// TwinCAT 3 PLC project Area2
// ProgramVersion: 3.1.4023.0
// libraries:
//   Tc2_DataExchange, * (Beckhoff Automation GmbH)
//   Tc2_MC2, * (Beckhoff Automation GmbH)
//   Tc2_Standard, * (Beckhoff Automation GmbH)
//   Tc2_System, * (Beckhoff Automation GmbH)
//   Tc2_TcpIp, * (Beckhoff Automation GmbH)
//   Tc2_Utilities, * (Beckhoff Automation GmbH)
//   Tc3_BA_Common, * (Beckhoff Automation GmbH)
//   Tc3_Database, * (Beckhoff Automation GmbH)
//   Tc3_JsonXml, * (Beckhoff Automation GmbH)
//   Tc3_Module, * (Beckhoff Automation GmbH)
//   Tc3_PackML_V2, * (Beckhoff Automation GmbH)
// project tree:
//   COMMs_ADS/ AdsClient.TcPOU, AdsHandle.TcPOU
//   COMMs_ADS/PROTOTYPE/ AdsClient_1.TcPOU, AdsHandle_1.TcPOU (not stored)
//   COMMs_TCP/ TcpServer1Vision.TcPOU (not stored)
//   COMMs_TCP/Types/ DUT.TcDUT (not stored), TcpData.TcDUT, TcpDataQueue.TcPOU (not stored)
//   DUTs/Enums/ E_PMLCustomUnitMode.TcDUT, InsertionDirection.TcDUT (not stored), SectionEnum.TcDUT (not stored), SectionTask.TcDUT, ConveyorMode.TcDUT (not stored), Cover.TcDUT, EventsEnum.TcTLEO (not stored), MaterialEnums.TcDUT (not stored), MaterialType.TcDUT, Surface.TcDUT (not stored)
//   DUTs/Enums/Materials/ Cardboard.TcDUT (not stored), Chipboard.TcDUT (not stored), CornerGuard.TcDUT (not stored), WoodBunk.TcDUT (not stored)
//   DUTs/Enums/Robot Tasks/ A22.TcDUT, A21.TcDUT
//   DUTs/Hardware/ A21ToolStorage.TcDUT (not stored), ConveyorLSC.TcPOU (not stored), ConveyorSC.TcPOU, FoldingMachine.TcDUT (not stored), Conveyor.TcPOU (not stored)
//   DUTs/Hardware/Big Machines/ StrapMachine.TcPOU, WrapMachine.TcPOU
//   DUTs/Hardware/Insertion Package/Drives/ AirPiston.TcPOU (not stored), ClearLinkMC.TcPOU (not stored), ServoNC.TcPOU (not stored), SimplePiston.TcPOU
//   DUTs/Hardware/Insertion Package/ Homing.TcDUT, Insertion.TcPOU, SuctionPad.TcDUT (not stored)
//   DUTs/Hardware/Insertion Package/Prototypes/ FBA_Drive.TcPOU, FBA_TrifectaDrive.TcPOU (not stored), I_ContinuousDrive.TcIO, I_Drive.TcIO (not stored), I_EncodedDrive.TcIO (not stored), I_PositionalDrive.TcIO
//   DUTs/Hardware/Material Holders/ MaterialHolder.TcPOU, MaterialSlot.TcDUT, SkidMagazine.TcPOU (not stored), StagingTable.TcPOU (not stored)
//   DUTs/Hardware/Robots/ KukaRobot.TcPOU, RobotA21.TcPOU, RobotA22.TcPOU
//   DUTs/ ONE_BIT.TcDUT (not stored), VisionFrame.TcDUT (not stored), VisionSuite.TcDUT (not stored)
//   COMMs_ADS/Types/ AdsSocket.TcPOU (not stored), AdsDataQueue.TcPOU (not stored), AdsData.TcDUT (not stored)
//   DUTs/Bundle/ Bundle.TcDUT, CardboardMaterial.TcDUT (not stored), Interval.TcDUT (not stored), Material.TcDUT (not stored), PositionMaterials.TcDUT (not stored)
//   DUTs/Containers/ DynamicQueue.TcPOU (not stored), PtrQueue.TcPOU (not stored), IntQueue.TcPOU, Queue.TcPOU (not stored), StringQueue.TcPOU
//   EventLogging/ EventLogger.TcIO (not stored), SqlDatabaseAccessor.TcPOU (not stored)
//   / GlobalTextList.TcGTLO, PlcTask.TcTTO (not stored)
//   GVLs/ Conveyors.TcGVL, GVL.TcGVL, Hardware_A21.TcGVL, Hardware_A22.TcGVL, Hardware_A23.TcGVL, Hardware_A24.TcGVL (not stored), Hardware_A25.TcGVL (not stored), Misc.TcGVL (not stored), Param.TcGVL
//   POUs/ CallHardware.TcPOU, ConveyorControlUnit.TcPOU, MAIN.TcPOU
//   POUs/Helper Functions/Document/ CreateJsonDocumentManual.TcPOU, CreateJsonDocumentAuto.TcPOU (not stored), FrameIsValid.TcPOU (not stored), VisionJsonParser.TcPOU (not stored)
//   POUs/Helper Functions/General/ BufferIsEmpty.TcPOU (not stored), BundleIsValid.TcPOU, InRange.TcPOU (not stored), PositionIsValid.TcPOU, TimestructToString.TcPOU (not stored)
//   POUs/Helper Functions/Hardware Modules/ InsertionQuality.TcPOU (not stored), SetSuctions.TcPOU (not stored), SetSuctionsPtrArr.TcPOU (not stored), SetupHardware.TcPOU, SuctionQuality.TcPOU (not stored)
//   POUs/Helper Functions/Material Functions/ GetPositionMasterLength.TcPOU (not stored), GetMaterialLength.TcPOU (not stored), MatchesMaterialType.TcPOU (not stored)
//   POUs/Helper Functions/Other/ ForceSetLifterConveyors.TcPOU (not stored), SizeCheck.TcPOU (not stored)
//   POUs/Helper Functions/Utility/ AddToStringArray.TcPOU (not stored), DataIsEmtpy.TcPOU, CleanStringsArray.TcPOU, IntegerBitAccess.TcPOU, IntegerToBoolArray.TcPOU (not stored), JoinStrings.TcPOU (not stored), WithinTolerance.TcPOU
//   Sections/A21a - Chipboard/AOIs/ AOI_LoadChipboard.TcPOU
//   Sections/A21a - Chipboard/ ChipboardEx.TcPOU
//   Sections/A21b - Wood Bunk/AOIs/ AOI_LoadWoodBunk.TcPOU, AOI_StageWoodBunk.TcPOU, AOI_StagingTemplate.TcPOU, AOI_WoodBunkAlarms.TcPOU (not stored)
//   Sections/A21b - Wood Bunk/ WoodBunkEx.TcPOU
//   Sections/Abstract/ SectionEx.TcPOU
// real-time tasks:
//   TASK PlcTask: cycle T#10ms, priority 20, ADS port 350

// ---- COMMs_TCP/Types/TcpData.TcDUT
{attribute 'enable_dynamic_creation'}
TYPE TcpData :
UNION
	binaryData : ARRAY[0..1000] OF BYTE; //contents
	toString : STRING(1000);
END_UNION
END_TYPE

// ---- DUTs/Enums/E_PMLCustomUnitMode.TcDUT
//{attribute 'qualified_only'}
//{attribute 'strict'}
TYPE E_PMLCustomUnitMode :
(
	ePMLCustomUnitMode_Invalid := 0, //no mode
	ePMLCustomUnitMode_Production := 1, //normal automatic production
	ePMLCustomUnitMode_Maintenance := 2, //testing operational improvements
	ePMLCustomUnitMode_Manual := 3, //commissioning
	
	ePMLCustomUnitMode_SemiAuto := 4, //same state machine as production, but uses an execute signal to advance to next step
	
	size
)DINT;
END_TYPE
(*
this enum adds on to E_PMLProtectedUnitMode with additional modes
can be used by a combobox on the HMI to select a mode

all modes used in the program need to be configured using PML_UnitModeConfig
*)

// ---- DUTs/Enums/Robot Tasks/A22.TcDUT
{attribute 'qualified_only'}
{attribute 'to_string'}
//{attribute 'strict'}
TYPE A22 :
(
	IDLE,
	
	LOAD_CARDBOARD_TOP, //flat cardboards
	LOAD_CARDBOARD_BOTTOM,
	LOAD_CARDBOARD_SIDE,
	REMOVE_CARDBOARD_TOP,
	REMOVE_CARDBOARD_BOTTOM,
	REMOVE_CARDBOARD_SIDE,
	
	TRANSFER_TO_BENDER := 9, //corner cardboards
	TRANSFER_TO_OVERHEAD,
	REMOVE_CARDBOARD_FROM_BENDER,
	LOAD_BENDER_TO_UPPER_CORNER,
	LOAD_BENDER_TO_LOWER_CORNER,
	LOAD_OVERHEAD_TO_UPPER_CORNER,
	LOAD_OVERHEAD_TO_LOWER_CORNER,
	
	REMOVE_CARDBOARD_UPPER_CORNER,
	REMOVE_CARDBOARD_LOWER_CORNER,
	REMOVE_CARDBOARD_OVERHEAD := 18,
	
	LOAD_CORNER_GUARD_UPPER := 20, //corner guards
	LOAD_CORNER_GUARD_LOWER,
	REMOVE_CORNER_GUARD_UPPER,
	REMOVE_CORNER_GUARD_LOWER,
	
	size
);
END_TYPE

// ---- DUTs/Hardware/Insertion Package/Homing.TcDUT
{attribute 'qualified_only'}
{attribute 'strict'}
TYPE Homing :
(
	IDLE,
	
	START,
	RETRY,
	
	STOP,
	SET,
	DONE,
	
	size
);
END_TYPE
(*
general homing sequence:
	on drive.homingSequence() call, home towards home sensor
	if home reached, set position and finish homing as usual
	if outer limit reached, traverse towards inner limit
		when inner limit reached, retry homing
*)

// ---- DUTs/Hardware/Material Holders/MaterialSlot.TcDUT
TYPE MaterialSlot :
STRUCT
	material : STRING;
	occupied AT %I* : BOOL;
END_STRUCT
END_TYPE

// ---- DUTs/Enums/Robot Tasks/A21.TcDUT
{attribute 'qualified_only'}
//{attribute 'strict'}
{attribute 'to_string'}
TYPE A21 :
(
	IDLE,
	STAGE_BUNK,
	REMOVE_BUNK_FROM_STAGE,
	
	LOAD_BUNK_TOP := 4,
	LOAD_BUNK_SIDE,
	LOAD_BUNK_BOTTOM,
	REMOVE_BUNK_TOP,
	REMOVE_BUNK_SIDE,
	REMOVE_BUNK_BOTTOM,
	
	//GET_CHIPBOARD_FROM_SKID := 11,
	//OFFLOAD_CHIPBOARD,
	PLACE_CHIPBOARD_TOP := 13,
	PLACE_CHIPBOARD_BOTTOM,
	REMOVE_CHIPBOARD_TOP,
	REMOVE_CHIPBOARD_BOTTOM,
	
	FIX_CHIPBOARD_ORIENTATION := 19,
	
	//testing only
	MOVE_HOME := 21,
	MOVE_POSITION1,
	MOVE_POSITION2,
	MOVE_UP,
	MOVE_DOWN,
	
	DIRECT_BUNK_TOP := 27,
	DIRECT_BUNK_SIDE,
	DIRECT_BUNK_BOTTOM,
	
	INSPECT_BUNK := 31,
	INSPECT_CHIPBOARD,
	
	TOOL_CHANGE_BUNK := 34,
	TOOL_CHANGE_CHIPBOARD,
	
	size
);
END_TYPE

// ---- DUTs/Bundle/Bundle.TcDUT
{attribute 'enable_dynamic_creation'}
TYPE Bundle :
STRUCT
	id : STRING;
	weight : REAL;
	
	length : INT;
	width : INT;
	height : INT;
	
	pieces : INT;
	layers : INT;
	piecesPerLayer : INT;
	
	extrusionWeight : INT;
	extrusionHeight : INT;
	extrusionWidth : INT;
	
	//if a process is true, send it to the correct area and turn it false when complete
	reqProcesses : ARRAY[0..3] OF BOOL;
	
	manRE, autoRE : BOOL; //repacking - coming soon
	manSS, autoSS : BOOL; //packaging
	
	currStep : USINT; //for runtime use only
	
	paperFront : BOOL;
	paperBack : BOOL;
	cardboardFront : BOOL;
	cardboardBack : BOOL;
	
	paperTop : ARRAY[0..GVL.maxPairs] OF Interval;
	paperLeft : ARRAY[0..GVL.maxPairs] OF Interval;
	paperRight : ARRAY[0..GVL.maxPairs] OF Interval;
	paperBottom : ARRAY[0..GVL.maxPairs] OF Interval;
		
	cardboard : ARRAY[0..GVL.maxPairs] OF PositionMaterials;
	cardboardFolds : ARRAY[Surface.TOP_LEFT..Surface.BOTTOM_RIGHT] OF ARRAY[0..GVL.maxPairs] OF INT;
	
	topLeftFolds : ARRAY[0..GVL.maxPairs] OF INT;
	topRightFolds : ARRAY[0..GVL.maxPairs] OF INT;
	bottomLeftFolds : ARRAY[0..GVL.maxPairs] OF INT;
	bottomRightFolds : ARRAY[0..GVL.maxPairs] OF INT;
	
	cornerGuard : ARRAY[0..GVL.maxPairs] OF PositionMaterials;
	
	chipboard : ARRAY[0..GVL.maxPairs] OF PositionMaterials;
	woodBunk : ARRAY[0..GVL.maxPairs] OF PositionMaterials;
	
	cardboard_over_cornerGuard : BOOL;
	
	//for production log database
	timeStart : TIMESTRUCT;
	timeDone : TIMESTRUCT;
END_STRUCT
END_TYPE

// ---- DUTs/Enums/SectionTask.TcDUT
{attribute 'qualified_only'}
//{attribute 'strict'}
TYPE SectionTask :
(
	IDLE,
	ALIGNING,
	ACTIVE,
	CLEARING,
	COMPLETE,
	
	size
);
END_TYPE

// ---- DUTs/Enums/Cover.TcDUT
{attribute 'qualified_only'}
{attribute 'strict'}
TYPE Cover :
(
	FRONT,
	BACK,
	size
);
END_TYPE

// ---- DUTs/Enums/MaterialType.TcDUT
{attribute 'qualified_only'}
{attribute 'strict'}
TYPE MaterialType :
(
	PAPER,
	CARDBOARD,
	CORNER_GUARD,
	CHIPBOARD,
	WOOD_BUNK,
	size
);
END_TYPE

// ---- GVLs/Conveyors.TcGVL
//{attribute 'qualified_only'}
VAR_GLOBAL CONSTANT
	numConveyors : INT := 38;
END_VAR
VAR_GLOBAL
	conveyorsArr : ARRAY[1..numConveyors] OF POINTER TO ConveyorSC;
	
	A24_LRC_C02 	: Conveyor; //these conveyoors move bundles from A2.7 to A2.4
	A24_LRC_C04 	: Conveyor;
	A24_LRC_C06	 	: Conveyor;
	A24_LRC_C08 	: Conveyor;
	A24_LRC_C10 	: Conveyor;
	A24_LRC_C12 	: Conveyor;
	
	A24_SC_C01 		: ConveyorSC; //these conveyors move bundles on A2.4 forward down the cell
	A24_SC_C03 		: ConveyorSC;
	A24_SC_C05 		: ConveyorSC;
	A24_SC_C07 		: ConveyorSC;
	A24_SC_C09 		: ConveyorSC;
	A24_SC_C11 		: ConveyorSC;
	A24_SC_C13 		: ConveyorSC;
	
	A23_LSC_C14 	: ConveyorLSC;
	
	A22_SC_C15 		: ConveyorSC;
	A22_LSC_C16 	: ConveyorLSC;
	A22_LSC_C17 	: ConveyorLSC;
	
	A21_SC_C18 		: ConveyorSC;
	A21_LSC_C19 	: ConveyorLSC;
	A21_LSC_C20 	: ConveyorLSC;
	A21_LSC_C21 	: ConveyorLSC;
	
	A25_SC_C22 		: ConveyorSC;
	A25_LSC_C23 	: ConveyorLSC;
	A25_SC_C24 		: ConveyorSC;
	A25_LSLCC_C25 	: ConveyorLSC;
	A25_SC_C26 		: ConveyorSC;
	A25_LSLCC_C27 	: ConveyorLSC;
	A25_SC_C28 		: ConveyorSC;
	A25_LSC_C29 	: ConveyorLSC;
	A25_SC_C30 		: ConveyorSC;
	
	A25_SC_C31 		: ConveyorSC; //these conveyors move the bundle sideways onto the output buffers
	A25_SC_C32 		: ConveyorSC;
	A25_SC_C33 		: ConveyorSC;
	A25_SC_C34 		: ConveyorSC;
	A25_SC_C35 		: ConveyorSC;
	A25_SC_C36 		: ConveyorSC;
	A25_SC_C37 		: ConveyorSC;
	A25_SC_C38 		: ConveyorSC;
END_VAR

// ---- GVLs/GVL.TcGVL
{attribute 'qualified_only'}
VAR_GLOBAL CONSTANT
	maxPairs : USINT := 16;
	initArraySize : USINT := 4;
	maxQueue : INT := 16;
	
	nullPos : REAL := -1;
	
	numMaterials : INT := 32;
	allMaterials : ARRAY[0..numMaterials] OF Material := [
		(code := 'PAP28', width := 28, length := -1),
		
		(code := 'CAR20S', width := 20, length := 30),
		(code := 'CAR20M', width := 20, length := 45),
		(code := 'CAR20L', width := 20, length := 60),
		(code := 'CAR28S', width := 28, length := 30),
		(code := 'CAR28M', width := 28, length := 45),
		(code := 'CAR28L', width := 28, length := 60),
		
		(code := 'COR48', width := 1.5, length := 48),
		(code := 'COR96', width := 1.5, length := 96),
		
		(code := 'CIP18', width := 20, length := 18),
		(code := 'CIP54', width := 20, length := 54),
		
		(code := 'WDT20', width := 20, length := 2.5),
		(code := 'WDT22', width := 22, length := 2.5),
		(code := 'WDT28', width := 28, length := 2.5),
		
		(code := 'WDB20', width := 20, length := 2.5),
		(code := 'WDB22', width := 22, length := 2.5),
		(code := 'WDB28', width := 28, length := 2.5),
		
		(code := 'WDS08', width := 8, length := 2.5),
		(code := 'WDS10', width := 10, length := 2.5),
		(code := 'WDS12', width := 12, length := 2.5),
		(code := 'WDS14', width := 14, length := 2.5),
		(code := 'WDS8x8', width := 16, length := 2.5),
		(code := 'WDS8x10', width := 18, length := 2.5),
		(code := 'WDS20', width := 20, length := 2.5),
		(code := 'WDS22', width := 22, length := 2.5),
		(code := 'WDS12x12', width := 24, length := 2.5),
		(code := 'WDS12x14', width := 26, length := 2.5),
		(code := 'WDS28', width := 28, length := 2.5),
		(code := 'WDS20x10', width := 30, length := 2.5),
		(code := 'WDS20x12', width := 32, length := 2.5),
		
		(code := 'WDW20', width := 20, length := 6),
		(code := 'WDW22', width := 22, length := 6)]; //+1 null material

	//nullBundle : Bundle;
	
	//conveyorLength : REAL := 0;
	precisionTolerance : REAL := 0.05 * 25.4;
END_VAR
VAR_GLOBAL
	bundleOut : Bundle; //may or may not be used?
END_VAR

// ---- GVLs/Hardware_A21.TcGVL
//{attribute 'qualified_only'}
VAR_GLOBAL
	robot1 : RobotA21;
	robot2 : RobotA21;
	
	toolStorageA21Left : A21ToolStorage;
	toolStorageA21Right : A21ToolStorage;
	
	skidA21Left : SkidMagazine;
	skidA21Right : SkidMagazine;
	
	magazineA21Left : SkidMagazine;
	magazineA21Right : SkidMagazine;
	stagingTableLeft : StagingTable;
	stagingTableRight : StagingTable;
	
	strapperA21 : StrapMachine;
	
	horizontalDriveA21Left, horizontalDriveA21Right : AirPiston := (
		limitSensorDefaultState := FALSE,
		useBrake := FALSE);
	
	verticalDriveA21Left, verticalDriveA21Right : ClearLinkMC := (
		limitSensorDefaultState := TRUE, 
		homingDirectionOut := TRUE, //outwards (up)
		minPosition := 0,
		displacementPerRotation := 1,
		unitsPerPulse := 8000); //0.1x gearbox, 10 revs/pulse to compensate
		
	insertionA21left : Insertion;
	insertionA21Right : Insertion;
	
	pistonA21Bottom : SimplePiston;
	
	suctionA21Top : ARRAY[1..3] OF SuctionPad;
	suctionA21Left : ARRAY[1..4] OF SuctionPad;
	suctionA21Right : ARRAY[1..4] OF SuctionPad; 
	suctionA21Bottom : ARRAY[1..2] OF SuctionPad;
END_VAR
VAR_GLOBAL

	skidHmiA21Left, skidHmiA21Right AT %M* : ARRAY[1..2] OF MaterialSlot;
	magazineHmiA21Left, magazineHmiA21Right AT %M* : ARRAY[1..15] OF MaterialSlot;
	tableHmiA21Left, tableHmiA21Right : ARRAY[1..10] OF MaterialSlot;
END_VAR

// ---- GVLs/Hardware_A22.TcGVL
//{attribute 'qualified_only'}
VAR_GLOBAL
	robot3 : RobotA22;
	robot4 : RobotA22;
	
	benderA22Left : FoldingMachine;
	
	skidA22Left : SkidMagazine;
	skidA22Right : SkidMagazine;
	magazineA22Left : SkidMagazine;
	magazineA22Right : SkidMagazine;
	
	wrapperA22 : WrapMachine;
	overhead : STRING;
	
	horizontalDriveA22Left, horizontalDriveA22Right : ServoNC := (
		limitSensorDefaultState := TRUE);
		
	verticalDriveA22Left, verticalDriveA22Right : ClearLinkMC := (
		limitSensorDefaultState := TRUE, 
		homingDirectionOut := TRUE, //outwards (up)
		minPosition := (26*5 * 25.4),
		displacementPerRotation := 5,
		unitsPerPulse := 800); //800 counts = 1 rotation
		
	insertionA22Left : Insertion;
	insertionA22Right : Insertion;

	pistonA22Bottom : SimplePiston;
	
	(*
	each insertion suction array has 3 pads
	[1] - top/bottom
	[2] - corner
	[3] - side
	*)
	suctionA22TopLeft : ARRAY[1..3] OF SuctionPad;
	suctionA22TopRight : ARRAY[1..3] OF SuctionPad;
	suctionA22BottomLeft : ARRAY[1..3] OF SuctionPad; 
	suctionA22BottomRight : ARRAY[1..3] OF SuctionPad;
	
	suctionA22Bottom : ARRAY[1..2] OF SuctionPad;
END_VAR
VAR_GLOBAL //data arrays to be passed into material holder FBs - do not access directly
	skidHmiA22Left, skidHmiA22Right AT %M* : ARRAY[1...Cardboard.size-1] OF MaterialSlot;
	magazineHmiA22Left, magazineHmiA22Right AT %M* : ARRAY[1..CornerGuard.size-1] OF MaterialSlot;
END_VAR

// ---- GVLs/Hardware_A23.TcGVL
//{attribute 'qualified_only'}
VAR_GLOBAL
	//robot5 : RobotA23;
	//robot6 : RobotA23;
	
	//6 ClearLinkMC
	//3 or 4 ServoNC
	
	wrapperA23 : WrapMachine;
END_VAR

// ---- GVLs/Param.TcGVL
{attribute 'qualified_only'}
VAR_GLOBAL CONSTANT
END_VAR

// ---- DUTs/Hardware/Insertion Package/Prototypes/I_ContinuousDrive.TcIO
INTERFACE I_ContinuousDrive EXTENDS I_Drive

METHOD ABSTRACT moveContinuous : BOOL
VAR_INPUT
	direction : MC_Direction;
END_VAR
END_METHOD

END_INTERFACE

// ---- DUTs/Hardware/Insertion Package/Prototypes/I_PositionalDrive.TcIO
INTERFACE I_PositionalDrive EXTENDS I_Drive

{attribute 'monitoring':='call'}
PROPERTY AtOuterLimit : BOOL
GET
END_GET
END_PROPERTY

PROPERTY CurrentPosition : LREAL
GET
END_GET
SET
END_SET
END_PROPERTY

METHOD ABSTRACT moveAbsolute : BOOL
VAR_INPUT
	newTarget : LREAL; 
END_VAR
END_METHOD

METHOD ABSTRACT moveRelative : BOOL
VAR_INPUT
	distance : LREAL;
END_VAR
END_METHOD

PROPERTY TargetPosition : LREAL
GET
END_GET
SET
END_SET
END_PROPERTY

END_INTERFACE

// ---- DUTs/Hardware/ConveyorSC.TcPOU
FUNCTION_BLOCK ConveyorSC
VAR_INPUT
	bEnable : BOOL;
END_VAR
VAR_OUTPUT
	trueMode : ConveyorMode;
	requestedMode : ConveyorMode;
	
	error AT %I* : BOOL;
	position AT %I* : REAL;
	velocity AT %I* : REAL;
END_VAR
VAR
	enable AT %Q* : BOOL := TRUE;
	direction AT %Q* : BOOL; //FALSE = forward, TRUE = backward
	pulse AT %Q* : BOOL;
	reset AT %Q* : BOOL;
	
	sensorEntry AT %I* : BOOL := TRUE;
	sensorExit AT %I* : BOOL;
END_VAR
VAR
	//nextConveyor : POINTER TO ConveyorSC;
	//prevConveyor : POINTER TO ConveyorSC;
	
	pulser : TP; //pulses are assumed to be low-high-low
END_VAR
VAR_STAT CONSTANT
	pulseWidth : TIME := T#50MS;
END_VAR

enable := bEnable;

override();

sequence();

METHOD backward : BOOL
VAR_INPUT
END_VAR
END_METHOD

METHOD forward : BOOL
VAR_INPUT
END_VAR
END_METHOD

{attribute 'monitoring' := 'call'}
PROPERTY IsOccupied : BOOL
GET
IsOccupied := sensorExit OR sensorEntry;
END_GET
END_PROPERTY

METHOD join : BOOL
VAR_INPUT
	conveyor : POINTER TO ConveyorSC;
END_VAR
//nextConveyor := conveyor;
//conveyor^.prevConveyor := THIS;
END_METHOD

METHOD PROTECTED override : BOOL
VAR_INPUT
END_VAR
END_METHOD

METHOD reset : BOOL
VAR_INPUT
END_VAR
position := 0;
velocity := velocity; //no change
END_METHOD

METHOD PROTECTED sequence : BOOL
VAR_INPUT
END_VAR
direction := (trueMode = ConveyorMode.BACKWARD); //set direction bit

pulser(IN:= , PT:= pulseWidth, Q=> pulse, ET=> );
pulser.IN := 
	enable AND 
	NOT error AND 
	NOT reset AND 
	(trueMode = ConveyorMode.FORWARD OR trueMode = ConveyorMode.BACKWARD)
	AND pulser.Q; //ends pulse itself
END_METHOD

METHOD setMode : BOOL
VAR_INPUT
	mode : ConveyorMode;
END_VAR
trueMode := mode;
END_METHOD

METHOD setRequest : BOOL
VAR_INPUT
	newRequest : ConveyorMode;
END_VAR
requestedMode := newRequest;
END_METHOD

METHOD target : BOOL
VAR_INPUT
	targetPosition : REAL;
END_VAR
END_METHOD

END_FUNCTION_BLOCK

// ---- DUTs/Hardware/Robots/RobotA21.TcPOU
FUNCTION_BLOCK RobotA21 EXTENDS KukaRobot
VAR_OUTPUT //from outputs array
	{warning disable C0195}
	taskID : A21;
	param1 : INT;
	param2 : INT;
	Xmm : INT;
	Ymm : INT;
	Zmm : INT;
	angle : INT;
	stagingOccupancy : INT;
	insertionSuctionStatus : INT;
	magazineStatus : INT; //unused
	inspectionValue : INT;
	
	strapSafetyOut : BOOL;
END_VAR
VAR_OUTPUT //from inputs array
	tool : SectionEnum := SectionEnum.WOOD_BUNK;
	suspendedMaterial : STRING;
	//gripper : EOAT := (id := SectionEnum.WOOD_BUNK, material := '');
	
	completedTask : A21;
	eoatDistance : INT;
	woodBunkAvailability : INT;
	chipboardAvailability : INT;
	materialAtHoldingPosition : INT;
	
	strapSafetyIn : BOOL;
END_VAR
VAR
	reservationEnum : SectionEnum;
	hmiTask : STRING;
	hmiTool : STRING;
END_VAR
(*
extends KukaRobot
assigns descriptive labels to each IO group from the array
additional section-specific methods to get/set IO groups
*)

(*
parameters - aliases to IO elements
command - full IO array
*)
{warning disable C0195}
SUPER^();

strapSafetyOut := NOT strapperA21.enable AND NOT strapperA21.execute;
outputs[8].15 := strapSafetyOut;

outputs[1] := taskID;
outputs[2] := param1;
outputs[3] := param2;
outputs[4] := Xmm;
outputs[5] := Ymm;
outputs[6] := Zmm;
outputs[7] := angle;
outputs[8] := stagingOccupancy;
outputs[9] := insertionSuctionStatus;
outputs[10] := magazineStatus;
outputs[11] := inspectionValue;

outputs[8].15 := strapSafetyOut;

refreshParameters();

reservationEnum := reservation;
IF reservationEnum = SectionEnum.NULL_SECTION THEN
	hmiReservation := 'N/A';
ELSE
	hmiReservation := TO_STRING(reservationEnum);
END_IF

hmiTask := TO_STRING(taskID);
hmiTool := TO_STRING(tool);

{attribute 'monitoring' := 'call'}
PROPERTY Busy : BOOL
GET
VAR
	//emptyOutput : ARRAY[1..50] OF INT;
END_VAR
//Busy stays TRUE until outputs are cleared AND completed task has elapsed
//Ready is always inverse of Busy
refreshParameters();

Busy := taskID <> 0 OR completedTask <> 0;
END_GET
END_PROPERTY

METHOD changeEOAT : BOOL
VAR_INPUT
	targetTool : SectionEnum;
END_VAR
setGroup(group := 1, value := A21.TOOL_CHANGE_CHIPBOARD);
setGroup(group := 1, value := A21.TOOL_CHANGE_BUNK);

changeEOAT := tool = targetTool;
END_METHOD

METHOD clearCommand : BOOL
VAR_INPUT
END_VAR
SUPER^.clearCommand();

refreshParameters();
END_METHOD

{attribute 'monitoring' := 'call'}
PROPERTY Done : BOOL
GET
refreshParameters();

Done :=
	completedTask = taskID AND
	taskID <> 0 AND
	completedTask <> 0;
END_GET
END_PROPERTY

{attribute 'monitoring' := 'call'}
PROPERTY HoldMaterial : STRING
GET
HoldMaterial := suspendedMaterial;
END_GET
SET
suspendedMaterial := HoldMaterial;
END_SET
END_PROPERTY

{attribute 'monitoring' := 'call'}
PROPERTY Ready : BOOL
GET
refreshParameters();

Ready := taskID = 0 AND completedTask = 0;
END_GET
END_PROPERTY

METHOD PRIVATE refreshParameters : BOOL
VAR_INPUT
END_VAR
{warning disable C0196}
taskID := outputs[1];
param1 := outputs[2];
param2 := outputs[3];
Xmm := outputs[4];
Ymm := outputs[5];
Zmm := outputs[6];
angle := outputs[7];
stagingOccupancy := outputs[8];
insertionSuctionStatus := outputs[9];
magazineStatus := outputs[10]; //unused
inspectionValue := outputs[11];

completedTask := inputs[1];
eoatDistance := inputs[2];
woodBunkAvailability := inputs[3];
chipboardAvailability := inputs[4];
materialAtHoldingPosition := inputs[5];
//robotEOAT := inputs[6];

strapSafetyIn := inputs[4].15;
END_METHOD

METHOD setGroup : BOOL
VAR_INPUT
	group : INT;
	value : INT;
END_VAR
SUPER^.setGroup(group := group, value := value);

refreshParameters();
END_METHOD

METHOD setParameters : BOOL
VAR_INPUT
	newTaskID : INT;
	newParam1 : INT;
	newParam2 : INT;
	newXmm : INT;
	newYmm : INT;
	newZmm : INT;
	newAngle : INT;
	newStagingOccupancy : INT;
	newInsertionSuctionStatus : INT;
	newMagazineStatus : INT; //unused
	newInspectionValue : INT;
END_VAR
VAR_INPUT
	strapSafety : BOOL;
END_VAR
setGroup(group := 1, value := newTaskID);
setGroup(group := 2, value := newParam1);
setGroup(group := 3, value := newParam2);
setGroup(group := 4, value := newXmm);
setGroup(group := 5, value := newYmm);
setGroup(group := 6, value := newZmm);
setGroup(group := 7, value := newAngle);

newStagingOccupancy.15 := strapSafety;
setGroup(group := 8, value := newStagingOccupancy);

setGroup(group := 9, value := newInsertionSuctionStatus);
setGroup(group := 10, value := newMagazineStatus);
setGroup(group := 11, value := newInspectionValue);

refreshParameters();
END_METHOD

END_FUNCTION_BLOCK

// ---- DUTs/Hardware/Robots/KukaRobot.TcPOU
FUNCTION_BLOCK KukaRobot
VAR_OUTPUT
	forceStop AT %Q* : BOOL;
	resetSignal AT %Q* : BOOL;
	
	offline AT %I* : BOOL;
	operational : BOOL;
	reservation : INT := SectionEnum.NULL_SECTION;
	
	error : BOOL;
	errId : DINT;
	
	outputs AT %Q* : ARRAY[1..50] OF WORD;
	inputs AT %I* : ARRAY[1..20] OF WORD;
END_VAR
VAR
	hmiReservation : STRING;
END_VAR
(*
generic KUKA robot with 50 WORD outputs and 20 WORD inputs
includes minimal diagnostics to detect if robot is offline
robots should always be reserved before sending a task
*)

operational := NOT offline;

error := offline; //add any addition conditions with OR

//{attribute 'monitoring' := 'variable'}
{attribute 'monitoring' := 'call'}
PROPERTY Busy : BOOL
GET
END_GET
END_PROPERTY

METHOD clearCommand : BOOL
VAR_INPUT
END_VAR
MEMSET(ADR(outputs), 0, SIZEOF(outputs));
END_METHOD

//{attribute 'monitoring' := 'variable'}
{attribute 'monitoring' := 'call'}
PROPERTY Done : BOOL
GET
END_GET
END_PROPERTY

METHOD eStop : BOOL
VAR_INPUT
END_VAR
forceStop := TRUE;
eStop := TRUE;
END_METHOD

METHOD fullCommand : BOOL
VAR_INPUT
	newOutputs : REFERENCE TO ARRAY[1..50] OF WORD;
END_VAR
//IF NOT Busy THEN
	//RETURN;
//END_IF

outputs := newOutputs;
fullCommand := Done;

(*
CASE step OF
	SEND_COMMAND: //wait 1 cycle
		outputs := newOutputs;
		step := WAIT;
		
	WAIT:
		IF done THEN
			(*	
			IF NOT reset() THEN
				RETURN;
			END_IF
			
			step := 0;
			*)
			setCommandAndWait := TRUE;
		END_IF
		
END_CASE
*)
END_METHOD

{attribute 'monitoring' := 'call'}
PROPERTY Ready : BOOL
GET
END_GET
END_PROPERTY

METHOD release : BOOL
VAR_INPUT
	sectionReservation : SectionEnum;
END_VAR
IF reservation = sectionReservation THEN
	reservation := SectionEnum.NULL_SECTION;
	release := TRUE;
END_IF
END_METHOD

METHOD reserve : BOOL
VAR_INPUT
	reserveRequest : SectionEnum;
END_VAR
(*
this method exists because chipboard and wood bunk operations use the same robot
both sections need to check if the robot is open to commands before use
*)
IF Reserved AND reservation = reserveRequest THEN
	reserve := TRUE;

ELSIF NOT Reserved THEN
	reservation := reserveRequest;
	reserve := TRUE;

END_IF
END_METHOD

{attribute 'monitoring' := 'call'}
PROPERTY Reserved : BOOL
GET
Reserved := reservation <> SectionEnum.NULL_SECTION;
END_GET
END_PROPERTY

METHOD reset : BOOL
//resetSignal := TRUE;
//done := FALSE;

MEMSET(ADR(outputs), 0, SIZEOF(outputs));
(*
IF ready AND completedTask = 0 THEN
	resetSignal := FALSE;
	reset := TRUE;
END_IF
*)
END_METHOD

METHOD resume : BOOL
VAR_INPUT
END_VAR
forceStop := FALSE;

resume := NOT error AND errId = 0;
END_METHOD

METHOD setGroup : BOOL
VAR_INPUT
	group : INT;
	value : INT;
END_VAR
{warning disable C0195}
outputs[group] := value;
END_METHOD

END_FUNCTION_BLOCK

// ---- DUTs/Hardware/Big Machines/StrapMachine.TcPOU
FUNCTION_BLOCK StrapMachine
VAR_INPUT
	bEnable : BOOL;
END_VAR
VAR_OUTPUT
	enable AT %Q* : BOOL;
	execute AT %Q* : BOOL;
	reset AT %Q* : BOOL;
	
	error AT %I* : BOOL;
	ready AT %I* : BOOL;
	//busy (*AT %I**) : BOOL;
	done AT %I* : BOOL;
	home AT %I* : BOOL;
	
	timeout : BOOL;
	
	atBundleLevel AT %I* : BOOL;
END_VAR
VAR	
	holdPost : TON;
	timeoutDelay : TON;
	resetDelay : TP;
	
	start : BOOL;
	step : (SETUP, RUN, WAIT);
END_VAR
VAR_STAT CONSTANT
	maxDelay : TIME := T#30S;
	pulseWidth : TIME := T#500MS;
END_VAR

holdPost(IN:= , PT:= pulseWidth, Q=> , ET=> );
timeoutDelay(IN:= (step > 0), PT:= maxDelay, Q=> timeout, ET=> );

resetDelay(IN:= error AND NOT resetDelay.Q , PT:= pulseWidth, Q=> , ET=> );
reset := resetDelay.Q AND (resetDelay.ET > resetDelay.PT/2);

IF timeoutDelay.Q THEN
	timeoutDelay.IN := FALSE;
	timeout := TRUE;
	//busy := FALSE;
	
	start := FALSE;
	step := SETUP;
END_IF

enable := bEnable AND robot1.strapSafetyIn AND robot2.strapSafetyIn;

CASE step OF
	SETUP:
		IF error THEN
			enable := FALSE;
			execute := FALSE;
			RETURN;
		END_IF
		
		IF start AND enable (*AND ready*) THEN //strapping does not start if error
			start := FALSE;
			step := RUN;
		END_IF
	
	RUN:
		IF NOT execute THEN
			execute := TRUE;
			RETURN; //keeps execute TRUE for at least 1 cycle
		END_IF
		
		IF execute AND NOT ready (*AND NOT home*) THEN
			execute := FALSE;
			step := WAIT;
		END_IF
		
	WAIT: //due to the use of DC motors instead of stepper motors in the machine, a short delay is required before next strap
		IF home THEN
			holdPost.IN := TRUE;
			execute := FALSE;
			enable := FALSE;
		END_IF
		
		IF holdPost.Q THEN
			holdPost.IN := FALSE;
			step := 0;
		END_IF
		
END_CASE

(*
executePulse(IN:= , PT:= pulseTime, Q=> , ET=> );
execute := executePulse.IN AND NOT executePulse.Q;

IF executePulse.Q THEN
	executePulse.IN := FALSE;
END_IF


resetPulse(IN:= , PT:= pulseTime, Q=> , ET=> );
StrapMachineST.reset := resetPulse.IN AND NOT resetPulse.Q;

IF resetPulse.Q THEN
	executePulse.IN := FALSE;
END_IF

ready := enable AND NOT execute AND NOT StrapMachineST.reset AND NOT error AND home;
*)

METHOD clear : BOOL
VAR_INPUT
END_VAR
(*
reset should be continuously called until machine returns evidence that it is ready again
machine is expected to not respond to reset signals if it is already in an idle state
*)
END_METHOD

METHOD strap : BOOL
VAR_INPUT
END_VAR
//IF ready AND NOT busy AND NOT error THEN
	//busy := TRUE;
	//start := TRUE;
	//strap := TRUE;
//END_IF

start := TRUE;
END_METHOD

END_FUNCTION_BLOCK

// ---- DUTs/Hardware/Insertion Package/Insertion.TcPOU
FUNCTION_BLOCK Insertion //2d insertion that combines a slider (alignment) and screw (push)
VAR_INPUT
	enable : BOOL;
END_VAR
VAR_INPUT //interface references to existing drives
	slider : I_EncodedDrive;
	screw : I_ContinuousDrive;
END_VAR
VAR_OUTPUT
	contact AT %I* : BOOL;
	
	active : BOOL;
	error : BOOL;
	home : BOOL;
	
	homingComplete : BOOL;
	
	sliderPos : LREAL;
END_VAR
(*
this FB encapsulates 2 drives into a generic insertion machine
both drives should be declared externally in Hardware GVL as a concrete FB
Insertion instance should be declared and called in module scope, with the drives from Hardware GVL passed in by Interface reference
*)

homingComplete := slider.HomeSet AND screw.HomeSet;

active := slider.Active OR screw.Active;
error := slider.Error OR screw.Error;
home := slider.AtHome AND screw.AtHome;

sliderPos := slider.CurrentPosition;

METHOD align : BOOL
VAR_INPUT
	targetPos : REAL;
END_VAR
slider.moveAbsolute(newTarget := targetPos);
END_METHOD

METHOD homingSequence : BOOL
VAR_INPUT
END_VAR
IF NOT slider.homeSet THEN
	slider.homingSequence();
END_IF

IF NOT screw.homeSet THEN
	screw.homingSequence();
END_IF

homingSequence := homingComplete;
END_METHOD

METHOD press : BOOL
VAR_INPUT
END_VAR
screw.moveContinuous(direction := MC_Negative_Direction);
END_METHOD

METHOD release : BOOL
VAR_INPUT
END_VAR
screw.moveContinuous(direction := MC_Positive_Direction);
END_METHOD

METHOD reset : BOOL
VAR_INPUT
END_VAR
slider.reset();
screw.reset();
END_METHOD

METHOD stop : BOOL
VAR_INPUT
END_VAR
screw.stop();
slider.stop();
END_METHOD

METHOD toHome : BOOL
VAR_INPUT
END_VAR
slider.toHome();
screw.toHome();

toHome := slider.AtHome AND screw.AtHome;
END_METHOD

METHOD traverse : BOOL
VAR_INPUT
	direction : MC_Direction;
END_VAR
slider.moveContinuous(direction := MC_Negative_Direction);
END_METHOD

END_FUNCTION_BLOCK

// ---- DUTs/Hardware/Insertion Package/Drives/SimplePiston.TcPOU
FUNCTION_BLOCK SimplePiston
VAR_INPUT
	bEnable : BOOL;
END_VAR
VAR_OUTPUT
	pistonExtend AT %Q* : BOOL;
	pistonRetract AT %Q* : BOOL;
	
	extended AT %I* : BOOL;
	retracted AT %I* : BOOL;
	
	busy : BOOL;
END_VAR
VAR
	mode : (HOLD, IN, OUT);
END_VAR

IF
	NOT bEnable OR
	(retracted AND_THEN (pistonRetract OR mode = OUT)) OR
	(extended AND_THEN (pistonExtend OR mode = IN))
THEN
	mode := HOLD;
END_IF

CASE mode OF
	HOLD:
		pistonRetract := FALSE;
		pistonExtend := FALSE;
		
	IN:
		pistonRetract := FALSE;
		pistonExtend := TRUE;
	
	OUT:
		pistonRetract := TRUE;
		pistonExtend := FALSE;
	
END_CASE

busy := mode = IN OR mode = OUT;

METHOD extend : BOOL
VAR_INPUT
END_VAR
mode := IN;
END_METHOD

METHOD retract : BOOL
VAR_INPUT
END_VAR
mode := OUT;

retract := retracted;
END_METHOD

METHOD stop : BOOL
VAR_INPUT
END_VAR
pistonExtend := FALSE;
pistonRetract := FALSE;
mode := HOLD;
END_METHOD

END_FUNCTION_BLOCK

// ---- DUTs/Hardware/Robots/RobotA22.TcPOU
FUNCTION_BLOCK RobotA22 EXTENDS KukaRobot
VAR_OUTPUT //from outputs array
	taskID : A22;
	param1 : INT;
	param2 : INT;
	Xmm : INT;
	Ymm : INT;
	Zmm : INT;
	angle : INT;
	foldPosition0 : INT;
	foldPosition1 : INT;
END_VAR
VAR_OUTPUT //from inputs array
	tool : SectionEnum := SectionEnum.CARDBOARD_CORNERGUARD;
	suspendedMaterial : STRING;
	
	completedTask : A22;
	eoatDistance : INT;
	cardboardAvailability : INT;
	cornerGuardAvailability : INT;
	materialAtHoldingPosition : INT;
	//grp6
	//grp7
	
	wrapSafetyIn : BOOL;
	
END_VAR
VAR //HMI data
	reservationEnum : SectionEnum;
	hmiTask : STRING;
	hmiTool : STRING;
END_VAR

{warning disable C0195}
SUPER^();

outputs[1] := taskID;
outputs[2] := param1;
outputs[3] := param2;
outputs[4] := Xmm;
outputs[5] := Ymm;
outputs[6] := Zmm;
outputs[7] := angle;
outputs[8] := foldPosition0;
outputs[9] := foldPosition1;

refreshParameters();

reservationEnum := reservation;
IF reservationEnum = SectionEnum.NULL_SECTION THEN
	hmiReservation := 'N/A';
ELSE
	hmiReservation := TO_STRING(reservationEnum);
END_IF

hmiTask := TO_STRING(taskID);
hmiTool := TO_STRING(tool);

{attribute 'monitoring' := 'call'}
PROPERTY Busy : BOOL
GET
VAR
	//emptyOutput : ARRAY[1..50] OF INT;
END_VAR
//Busy stays TRUE until outputs are cleared AND completed task has elapsed
//Ready is always inverse of Busy
refreshParameters();

Busy := taskID <> 0 OR completedTask <> 0;
END_GET
END_PROPERTY

METHOD changeEOAT : BOOL
VAR_INPUT
	targetTool : SectionEnum;
END_VAR
//fill in IO here

changeEOAT := TRUE;
END_METHOD

METHOD clearCommand : BOOL
VAR_INPUT
END_VAR
SUPER^.clearCommand();

refreshParameters();
END_METHOD

{attribute 'monitoring' := 'call'}
PROPERTY Done : BOOL
GET
refreshParameters();

Done :=
	completedTask = taskID AND
	taskID <> 0 AND
	completedTask <> 0;
END_GET
END_PROPERTY

{attribute 'monitoring' := 'call'}
PROPERTY HoldMaterial : STRING
GET
HoldMaterial := suspendedMaterial;
END_GET
SET
suspendedMaterial := HoldMaterial;
END_SET
END_PROPERTY

{attribute 'monitoring' := 'call'}
PROPERTY Ready : BOOL
GET
refreshParameters();

Ready := taskID = 0 AND completedTask = 0;
END_GET
END_PROPERTY

METHOD PRIVATE refreshParameters : BOOL
VAR_INPUT
END_VAR
{warning disable C0196}
taskID := outputs[1];
param1 := outputs[2];
param2 := outputs[3];
Xmm := outputs[4];
Ymm := outputs[5];
Zmm := outputs[6];
angle := outputs[7];
foldPosition0 := outputs[8];
foldPosition1 := outputs[9];

completedTask := inputs[1];
(*
eoatDistance := inputs[2];
magazineAvailability := inputs[3];
chipboardSkidInPosition := inputs[4];
materialAtHoldingPosition := inputs[5];
//robotEOAT := inputs[6];

strapSafetyIn := inputs[4].15;
*)
END_METHOD

METHOD setGroup : BOOL
VAR_INPUT
	group : INT;
	value : INT;
END_VAR
SUPER^.setGroup(group := group, value := value);

refreshParameters();
END_METHOD

METHOD setParameters : BOOL
VAR_INPUT
	newTaskID : INT;
	newParam1 : INT;
	newParam2 : INT;
	newXmm : INT;
	newYmm : INT;
	newZmm : INT;
	newAngle : INT;
	newStagingOccupancy : INT;
	newInsertionSuctionStatus : INT;
	newMagazineStatus : INT; //unused
	newInspectionValue : INT;
END_VAR
setGroup(group := 1, value := newTaskID);
setGroup(group := 2, value := newParam1);
setGroup(group := 3, value := newParam2);
setGroup(group := 4, value := newXmm);
setGroup(group := 5, value := newYmm);
setGroup(group := 6, value := newZmm);
setGroup(group := 7, value := newAngle);

newStagingOccupancy.15 := NOT wrapperA22.enable AND NOT wrapperA22.execute;
setGroup(group := 8, value := newStagingOccupancy);

setGroup(group := 9, value := newInsertionSuctionStatus);
setGroup(group := 10, value := newMagazineStatus);
setGroup(group := 11, value := newInspectionValue);

refreshParameters();
END_METHOD

END_FUNCTION_BLOCK

// ---- DUTs/Hardware/Big Machines/WrapMachine.TcPOU
FUNCTION_BLOCK WrapMachine
VAR_OUTPUT
	error AT %I* : BOOL;
	ready AT %I* : BOOL;
	busy AT %I* : BOOL;
	done (*AT %I**) : BOOL;
	home AT %I* : BOOL;
	
	rotations AT %Q* : INT;
	execute AT %Q* : BOOL;
	enable AT %Q* : BOOL;
	reset AT %Q* : BOOL;
	
	timeout : BOOL;
	
	trayOccupied AT %I* : BOOL;
	overheadMaterial : STRING;
END_VAR
VAR
	holdPost : TON;
	delay : TON;
	
	start : BOOL;
	step : (SETUP, RUN, WAIT);
END_VAR
VAR_STAT CONSTANT
	pulseTime : TIME := T#100MS;
	holdTime : TIME := T#500MS;
	maxDelay : TIME := T#30S;
END_VAR

holdPost(IN:= , PT:= holdTime, Q=> , ET=> );
delay(IN:= step > 0, PT:= maxDelay, Q=> , ET=> );

IF delay.Q THEN
	delay.IN := FALSE;
	timeout := TRUE;
	busy := FALSE;
	step := SETUP;
END_IF

CASE step OF
	SETUP:
		busy := FALSE;
		IF error THEN
			reset := NOT reset;
			enable := FALSE;//NOT enable;
			
		ELSE
			reset := FALSE;
			enable := TRUE;
			
			IF start THEN
				start := FALSE;
				step := RUN;
			END_IF
			
		END_IF
	
	RUN:
		execute := TRUE;
		IF execute AND NOT home THEN
			execute := FALSE;
			step := WAIT;
		END_IF
		
	WAIT:
		IF home THEN
			holdPost.IN := TRUE;
			enable := FALSE;
			execute := FALSE;
		END_IF
		
		IF holdPost.Q THEN
			holdPost.IN := FALSE;
			done := TRUE;
			step := 0;
		END_IF
		
END_CASE

METHOD clear : BOOL
VAR_INPUT
END_VAR
(*
reset should be continuously called until machine returns evidence that it is ready again
machine is expected to not respond to reset signals if it is already in an idle state
*)
enable := FALSE;
execute := FALSE;

IF error THEN
	reset := NOT reset;
	clear := NOT error;

ELSE
	reset := FALSE;
	clear := TRUE;
	
END_IF
END_METHOD

{attribute 'monitoring' := 'call'}
PROPERTY Overhead : STRING
GET
Overhead := overheadMaterial;
END_GET
SET
overheadMaterial := Overhead;
END_SET
END_PROPERTY

METHOD wrap : BOOL
VAR_INPUT
	reqRotations : INT;
END_VAR
IF ready AND NOT busy AND NOT error THEN
	rotations := reqRotations;
	busy := TRUE;
	start := TRUE;
	wrap := TRUE;
END_IF
END_METHOD

END_FUNCTION_BLOCK

// ---- COMMs_ADS/AdsClient.TcPOU
PROGRAM AdsClient
VAR_INPUT
	ServerNetId			: STRING; 	(* Server AmsNetId *)
	ServerPort 			: UINT;	(* Server port number *)
END_VAR
VAR_OUTPUT
	bBusy				: BOOL;
	err					: BOOL;
	errid				: UDINT;
	
	localPrgName 		: STRING;
	localNetId 			: STRING;
	localPort 			: UINT;
	
	socketReady				: BOOL;
	
	remoteAccessPrefix	: STRING := 'AdsServer.area[2].';
END_VAR
VAR
	setupTimer 			: TON;
	
	handle 				: AdsHandle;
	numHandles 			: INT(0..maxHandles);
	
	setupStep 			: (SET_LOCAL_ENDPOINT, CLOSE_CONNECTIONS, SEND_CONNECTION_DATA, RECEIVE_SERVER_DATA, FINISH_SETUP);
	
	fbGetLocalAmsNetId	: FB_GetLocalAmsNetId;
	
	i : INT;
	adsCtr : INT;
END_VAR
VAR CONSTANT
	maxHandles			: INT := 6;
END_VAR

socketReady := setup();
IF NOT socketReady THEN //setup after initialization
	RETURN;
END_IF

handle(
	ServerNetId:= ServerNetId,
	ServerPort:= ServerPort,
	
	remoteAccessPrefix := remoteAccessPrefix,
	
	bBusy=> bBusy,
	err=> err,
	errId=> errId,
	
	receiveBuffer=> ,
	receiveStruct=> );

METHOD fetchData : BOOL
VAR_IN_OUT
	receiverStruct : AdsData;
END_VAR
VAR
	emptyData : AdsData;
END_VAR
receiverStruct := handle.receiveStruct;

fetchData := MEMCMP(ADR(receiverStruct), ADR(emptyData), SIZEOF(AdsData)) <> 0; //returns false if no data

handle.clearBuffer();
END_METHOD

METHOD PROTECTED findHandle : REFERENCE TO AdsHandle
VAR_INPUT
	remotePrgName : STRING;
END_VAR
IF handle.getHandlerName() = remotePrgName THEN
	findHandle REF= handle;
	RETURN;
END_IF
END_METHOD

METHOD queueData : BOOL
VAR_INPUT
	data : REFERENCE TO AdsData;
END_VAR
handle.queueData(data);
END_METHOD

METHOD PROTECTED read : BOOL
VAR_INPUT
	remotePrgName : STRING;
	symbol : STRING;
	buffer : PVOID;
	symbolSize : UDINT;
END_VAR
VAR
	targetHandler : REFERENCE TO AdsHandle;
END_VAR
targetHandler REF= findHandle(remotePrgName);

IF __ISVALIDREF(targetHandler) THEN
	targetHandler.read(symbol, buffer, symbolSize);
END_IF
END_METHOD

METHOD PROTECTED send : BOOL
VAR_INPUT
	data : PVOID;
	dataSize : UDINT;
END_VAR
write(CONCAT(remoteAccessPrefix, 'genericBuffer'), data, dataSize);
END_METHOD

METHOD PROTECTED setup : BOOL
VAR
	pass : BOOL;
END_VAR
CASE setupStep OF
	SET_LOCAL_ENDPOINT:
		localPrgName := 'AREA_2';
		localPort := 851;
		
		fbGetLocalAmsNetId(
			bExecute:= , 
			tTimeOut:= , 
			bBusy=> , 
			bError=> , 
			nErrId=> , 
			AddrString=> localNetId, 
			AddrBytes=> );
		fbGetLocalAmsNetId.bExecute := NOT fbGetLocalAmsNetId.bExecute;	
		
		IF
			localPrgName <> '' AND
			localNetId <> '' AND localNetId <> '0.0.0.0.0.0' OR
			localPort <> 0
		THEN
			fbGetLocalAmsNetId.bExecute := FALSE;
			handle.open(localPrgName, localNetId, localPort);
			
			setupStep := CLOSE_CONNECTIONS;
		END_IF
		
	CLOSE_CONNECTIONS:
		handle.close();
		setupStep := SEND_CONNECTION_DATA;
		
	SEND_CONNECTION_DATA:
		CASE adsCtr OF
			0:
				pass := handle.write(
					symbol:= 'AdsServer.handle[1].socket.remotePrgName',
					data:= ADR(localPrgName),
					dataSize:= SIZEOF(localPrgName));
			
			1:
				pass := handle.write(
					symbol:= 'AdsServer.handle[1].socket.remoteNetId',
					data:= ADR(localNetId),
					dataSize:= SIZEOF(localNetId));
			
			2:
				pass := handle.write(
					symbol:= 'AdsServer.handle[1].socket.remotePort',
					data:= ADR(localPort),
					dataSize:= SIZEOF(localPort));
			
			3:
				adsCtr := 0;
				setupStep := RECEIVE_SERVER_DATA;
				RETURN;
			
		END_CASE
		
		IF pass THEN
			adsCtr := adsCtr + 1;
		END_IF
		
	RECEIVE_SERVER_DATA:
		CASE adsCtr OF
			0:
				pass := handle.read(
					symbol:= 'AdsServer.handle[2].socket.localPrgName', 
					buffer:= ADR(handle.socket.remotePrgName), 
					symbolSize:= SIZEOF(handle.socket.remotePrgName));
			
			1:
				pass := handle.read(
					symbol:= 'AdsServer.handle[2].socket.localNetId', 
					buffer:= ADR(handle.socket.remoteNetId), 
					symbolSize:= SIZEOF(handle.socket.remoteNetId));
			
			2:
				pass := handle.read(
					symbol:= 'AdsServer.handle[2].socket.localPort', 
					buffer:= ADR(handle.socket.remotePort), 
					symbolSize:= SIZEOF(handle.socket.remotePort));
			
			3:
				adsCtr := 0;
				setupStep := FINISH_SETUP;
				RETURN;
			
		END_CASE
		
		IF pass THEN
			adsCtr := adsCtr + 1;
		END_IF
			
	FINISH_SETUP:
		setup := TRUE;
		RETURN;
END_CASE
END_METHOD

METHOD PROTECTED write : BOOL
VAR
	remotePrgName : STRING := handle.socket.remotePrgName;
END_VAR
VAR_INPUT
	symbol : STRING;
	data : PVOID;
	dataSize : UDINT;
END_VAR
VAR
	targetHandle : REFERENCE TO AdsHandle;
END_VAR
targetHandle REF= findHandle(remotePrgName);

IF __ISVALIDREF(targetHandle) THEN
	targetHandle.write(symbol, data, dataSize);
END_IF
END_METHOD

END_PROGRAM

// ---- COMMs_ADS/AdsHandle.TcPOU
FUNCTION_BLOCK AdsHandle
VAR_INPUT
	ServerNetId			: STRING; 	(* Server AmsNetId *)
	ServerPort 			: UDINT;	(* Server port number *)
	
	remoteAccessPrefix	: STRING;
END_VAR
VAR_OUTPUT
	bBusy				: BOOL;
	err					: BOOL;
	errid				: UDINT;
	
	receiveBuffer		: ARRAY[0..100000] OF BYTE; //TCP style data buffer
	receiveStruct		: AdsData;
END_VAR
VAR	
	socket 				: AdsSocket; //only this needs initialization
	
	sendQueue			: AdsDataQueue;
	sendBufferQueue 	: DynamicQueue; //anything going into this needs to be a TcpStruct
	
	sendBuffer 			: ARRAY[0..50000] OF BYTE; //temp byte buffer to send if neccessary
	sendStruct			: AdsData;
	
	//setupStep 			: (CLOSE_CONNECTIONS, CREATE_LISTENER, ACCEPT_CONNECTION, FINISH_SETUP);
	sendDelay : TON;
END_VAR
VAR_STAT CONSTANT
	sendDelayTime : TIME := T#1S;
END_VAR

sendDelay(IN:= , PT:= sendDelayTime, Q=> , ET=> );
sendDelay.IN := TRUE;

IF sendDelay.Q THEN
	
	sendStruct := sendQueue.poll();
	IF NOT DataIsEmtpy(arr := ADR(sendStruct), arrSize := SIZEOF(sendStruct)) THEN //if valid data to send	
		write(
			symbol := CONCAT(remoteAccessPrefix, 'receiveStruct'),
			data := ADR(sendStruct),
			dataSize := SIZEOF(sendStruct));
			
		sendDelay.IN := FALSE;
	END_IF
	
END_IF

METHOD clearBuffer : BOOL
VAR
	emptyReceiverStruct : AdsData;
END_VAR
//MEMSET(ADR(receiveBuffer), 0, SIZEOF(receiveBuffer));
receiveStruct := emptyReceiverStruct;
END_METHOD

METHOD close : BOOL
VAR_INPUT
END_VAR
socket.close();
END_METHOD

METHOD getHandlerName : STRING
getHandlerName := socket.remotePrgName;
END_METHOD

METHOD open : BOOL
VAR_INPUT
	localPrgName : STRING;
	localNetId : T_AmsNetId;
	localPort : T_AmsPort;
END_VAR
socket.open(localPrgName, localNetId, localPort);
END_METHOD

METHOD queueData : BOOL
VAR_INPUT
	data : REFERENCE TO AdsData;
END_VAR
//MEMCPY(ADR(temp), data.pValue, data.diSize);
sendQueue.push(data);
END_METHOD

METHOD read : BOOL
VAR_INPUT
	symbol : STRING;
	buffer : PVOID;
	symbolSize : UDINT;
END_VAR
IF NOT socket.readBusy THEN
	read := socket.read(
		symbol:= symbol,
		buffer := buffer,
		symbolSize := symbolSize);
END_IF
END_METHOD

METHOD write : BOOL
VAR_INPUT
	symbol : STRING;
	data : PVOID;
	dataSize : UDINT;
END_VAR
VAR
	timer : TON;
END_VAR
IF NOT socket.writeBusy THEN
	write := socket.write(
		symbol:= symbol,
		data := data,
		dataSize := dataSize);
END_IF
END_METHOD

END_FUNCTION_BLOCK

// ---- POUs/Helper Functions/Utility/DataIsEmtpy.TcPOU
FUNCTION DataIsEmtpy : BOOL
VAR_INPUT
	arr : POINTER TO BYTE;
	arrSize : ULINT;
END_VAR
VAR
	i : ULINT;
END_VAR

FOR i:=0 TO arrSize-1 BY 1 DO
	IF arr[i] <> 0 THEN
		RETURN;
	END_IF
END_FOR

DataIsEmtpy := TRUE;

END_FUNCTION

// ---- COMMs_ADS/PROTOTYPE/AdsClient_1.TcPOU
PROGRAM AdsClient_1
VAR_OUTPUT
	ServerPrgName		: STRING;
	ServerNetId			: STRING; 	(* Server AmsNetId *)
	ServerPort 			: UINT;		(* Server port number *)
	
	LocalPrgName		: STRING;// := 'AREA_2';
	LocalNetId			: STRING;
	LocalPort			: UINT;// := 851;

	bBusy				: BOOL;
	err					: BOOL;
	errId				: UDINT;
	
	socketReady			: BOOL;
	
	remoteAccessPrefix	: STRING := 'AdsServer.area[2].';
END_VAR
VAR
	setupTimer 			: TON;
	
	handle				: AdsHandle_1;
	numHandles 			: INT(0..maxHandles);
	
	setupStep 			: (SET_LOCAL_ENDPOINT, CLOSE_CONNECTIONS, SEND_CONNECTION_DATA, RECEIVE_SERVER_DATA, FINISH_SETUP);
	
	fbGetLocalAmsNetId	: FB_GetLocalAmsNetId;
END_VAR
VAR CONSTANT
	maxHandles			: INT := 6;
END_VAR

socketReady := setup();

IF NOT socketReady THEN //setup after initialization
	RETURN;
END_IF
	
handle(
	RemotePrgName=> ServerPrgName, 
	RemoteNetId=> ServerNetId, 
	RemotePort=> ServerPort, 
	LocalPrgName=> LocalPrgName, 
	LocalNetId=> LocalNetId, 
	LocalPort=> LocalPort, 
	remoteAccessPrefix=> , 
	busy=> , 
	error=> , 
	errorId=> , 
	receiveBuffer=> , 
	receiveStruct=> );

METHOD fetchData : BOOL
VAR_IN_OUT
	receiverStruct : AdsData;
END_VAR
VAR
	emptyData : AdsData;
END_VAR
receiverStruct := handle.receiveStruct;

fetchData := MEMCMP(ADR(receiverStruct), ADR(emptyData), SIZEOF(AdsData)) <> 0; //returns false if no data

handle.clearBuffer();
END_METHOD

METHOD PROTECTED findHandle : REFERENCE TO AdsHandle
VAR_INPUT
	remotePrgName : STRING;
END_VAR
IF handle.getHandlerName() = remotePrgName THEN
	findHandle REF= handle;
	RETURN;
END_IF
END_METHOD

METHOD queueData : BOOL
VAR_INPUT
	data : REFERENCE TO AdsData;
END_VAR
handle.queueData(data);
END_METHOD

METHOD PROTECTED read : BOOL
VAR_INPUT
	remotePrgName : STRING;
	symbol : STRING;
	buffer : PVOID;
	symbolSize : UDINT;
END_VAR
VAR
	targetHandler : REFERENCE TO AdsHandle;
END_VAR
targetHandler REF= findHandle(remotePrgName);

IF __ISVALIDREF(targetHandler) THEN
	targetHandler.read(symbol, buffer, symbolSize);
END_IF
END_METHOD

METHOD PROTECTED send : BOOL
VAR_INPUT
	data : PVOID;
	dataSize : UDINT;
END_VAR
write(CONCAT(remoteAccessPrefix, 'genericBuffer'), data, dataSize);
END_METHOD

METHOD PROTECTED setup : BOOL
VAR
	pass : BOOL;
END_VAR
fbGetLocalAmsNetId(
	bExecute:= , 
	tTimeOut:= , 
	bBusy=> , 
	bError=> , 
	nErrId=> , 
	AddrString=> LocalNetId, 
	AddrBytes=> );
fbGetLocalAmsNetId.bExecute := NOT fbGetLocalAmsNetId.bExecute;

LocalPrgName := 'AREA_2';
LocalPort := 851;

handle.setup();




(*
IF
	localPrgName <> '' AND
	localNetId <> '' AND localNetId <> '0.0.0.0.0.0' AND
	localPort <> 0
THEN
	fbGetLocalAmsNetId.bExecute := FALSE;
	handle.open(localPrgName, localNetId, localPort);
	
	setupStep := CLOSE_CONNECTIONS;
END_IF

handle.setup();
*)
(*
CASE setupStep OF
	SET_LOCAL_ENDPOINT:
		localPrgName := 'AREA_2';
		localPort := 851;
		
		fbGetLocalAmsNetId(
			bExecute:= , 
			tTimeOut:= , 
			bBusy=> , 
			bError=> , 
			nErrId=> , 
			AddrString=> localNetId, 
			AddrBytes=> );
		fbGetLocalAmsNetId.bExecute := NOT fbGetLocalAmsNetId.bExecute;	
		
		IF
			localPrgName <> '' AND
			localNetId <> '' AND localNetId <> '0.0.0.0.0.0' OR
			localPort <> 0
		THEN
			fbGetLocalAmsNetId.bExecute := FALSE;
			handle.open(localPrgName, localNetId, localPort);
			
			setupStep := CLOSE_CONNECTIONS;
		END_IF
		
	CLOSE_CONNECTIONS:
		handle.close();
		setupStep := SEND_CONNECTION_DATA;
		
	SEND_CONNECTION_DATA:
		CASE adsCtr OF
			0:
				pass := handle.write(
					symbol:= 'AdsServer.handle[1].remotePrgName',
					data:= ADR(localPrgName),
					dataSize:= SIZEOF(localPrgName));
			
			1:
				pass := handle.write(
					symbol:= 'AdsServer.handle[1].remoteNetId',
					data:= ADR(localNetId),
					dataSize:= SIZEOF(localNetId));
			
			2:
				pass := handle.write(
					symbol:= 'AdsServer.handle[1].remotePort',
					data:= ADR(localPort),
					dataSize:= SIZEOF(localPort));
			
			3:
				adsCtr := 0;
				setupStep := RECEIVE_SERVER_DATA;
				RETURN;
			
		END_CASE
		
		IF pass THEN
			adsCtr := adsCtr + 1;
		END_IF
		
	RECEIVE_SERVER_DATA:
		CASE adsCtr OF
			0:
				pass := handle.read(
					symbol:= 'AdsServer.handle[2].socket.localPrgName', 
					buffer:= ADR(handle.socket.remotePrgName), 
					symbolSize:= SIZEOF(handle.socket.remotePrgName));
			
			1:
				pass := handle.read(
					symbol:= 'AdsServer.handle[2].socket.localNetId', 
					buffer:= ADR(handle.socket.remoteNetId), 
					symbolSize:= SIZEOF(handle.socket.remoteNetId));
			
			2:
				pass := handle.read(
					symbol:= 'AdsServer.handle[2].socket.localPort', 
					buffer:= ADR(handle.socket.remotePort), 
					symbolSize:= SIZEOF(handle.socket.remotePort));
			
			3:
				adsCtr := 0;
				setupStep := FINISH_SETUP;
				RETURN;
			
		END_CASE
		
		IF pass THEN
			adsCtr := adsCtr + 1;
		END_IF
			
	FINISH_SETUP:
		setup := TRUE;
		RETURN;
END_CASE
*)
END_METHOD

METHOD PROTECTED write : BOOL
VAR
	remotePrgName : STRING := handle.socket.remotePrgName;
END_VAR
VAR_INPUT
	symbol : STRING;
	data : PVOID;
	dataSize : UDINT;
END_VAR
VAR
	targetHandle : REFERENCE TO AdsHandle;
END_VAR
targetHandle REF= findHandle(remotePrgName);

IF __ISVALIDREF(targetHandle) THEN
	targetHandle.write(symbol, data, dataSize);
END_IF
END_METHOD

END_PROGRAM

// ---- DUTs/Hardware/Insertion Package/Prototypes/FBA_Drive.TcPOU
FUNCTION_BLOCK ABSTRACT FBA_Drive IMPLEMENTS I_Drive
VAR_INPUT
	bEnable : BOOL;
END_VAR
VAR //constructor
	limitSensorDefaultState : BOOL;
	//when a traverse sensor is opposite of this value, the respective property becomes TRUE
	//all sensors for a drive should be of the same type - do not mix & match PNP and NPN sensors on the same drive
END_VAR
VAR		
	homingComplete : BOOL;
	step : Homing;
	
	innerLimit AT %I* : BOOL; //replacable with homeLimit
	home AT %I* : BOOL;
	//not all drives have a rear limit, drives that do must extend from FBA_TrifectaDrive
END_VAR
(*
this abstract FB only specifies the minimum data for any drive
*)

{attribute 'monitoring':='call'}
PROPERTY ABSTRACT Active : BOOL
GET
END_GET
END_PROPERTY

{attribute 'monitoring':='call'}
PROPERTY AtHome : BOOL
GET
AtHome := home <> limitSensorDefaultState;
END_GET
END_PROPERTY

{attribute 'monitoring':='call'}
PROPERTY AtInnerLimit : BOOL
GET
AtInnerLimit := innerLimit <> limitSensorDefaultState;
END_GET
END_PROPERTY

{attribute 'monitoring':='call'}
PROPERTY ABSTRACT Error : BOOL
GET
END_GET
END_PROPERTY

{attribute 'monitoring':='call'}
PROPERTY HomeSet : BOOL
GET
HomeSet := homingComplete;
END_GET
END_PROPERTY

{attribute 'TcRpcEnable'}
METHOD ABSTRACT homingSequence : BOOL
VAR_INPUT
END_VAR
END_METHOD

{attribute 'TcRpcEnable'}
METHOD ABSTRACT reset : BOOL
VAR_INPUT
END_VAR
END_METHOD

{attribute 'TcRpcEnable'}
METHOD ABSTRACT stop : BOOL
VAR_INPUT
END_VAR
END_METHOD

METHOD ABSTRACT toHome : BOOL
VAR_INPUT
END_VAR
END_METHOD

END_FUNCTION_BLOCK

// ---- DUTs/Hardware/Material Holders/MaterialHolder.TcPOU
FUNCTION_BLOCK MaterialHolder
VAR_IN_OUT
	slots : ARRAY[*] OF MaterialSlot;
END_VAR
VAR_OUTPUT
	numSlots : INT;
END_VAR

numSlots := TO_INT(UPPER_BOUND(slots, 1) - LOWER_BOUND(slots, 1) + 1);

METHOD clear : BOOL
VAR_INPUT
END_VAR
VAR
	i : DINT;
END_VAR
FOR i:=LOWER_BOUND(slots, 1) TO UPPER_BOUND(slots, 1) BY 1 DO
	slots[i].material := '';
END_FOR
END_METHOD

METHOD compareWith : BOOL
VAR_INPUT
	src : REFERENCE TO MaterialHolder;
END_VAR
VAR
	i : DINT;
	j : DINT;
END_VAR
IF numSlots <> src.numSlots THEN
	RETURN;
END_IF

FOR i:=LOWER_BOUND(slots, 1) TO UPPER_BOUND(slots, 1) BY 1 DO //iterate through this instance's slots
	
	IF getSlot(i:= i, occupancy=> , error=> ) <> src.getSlot(i:= j, occupancy=> , error=> ) THEN
		RETURN;
	END_IF

END_FOR

compareWith := TRUE;
END_METHOD

METHOD copyFrom : BOOL
VAR_INPUT
	src : REFERENCE TO MaterialHolder;
END_VAR
VAR
	i : DINT;
	j : DINT;
END_VAR
j := LOWER_BOUND(src.slots, 1);

FOR i:=LOWER_BOUND(slots, 1) TO UPPER_BOUND(slots, 1) BY 1 DO //iterate through this instance's slots
	
	IF j <= UPPER_BOUND(src.slots, 1) THEN //if within bounds of src instance's slots
		slots[i].material := src.slots[j].material;
	END_IF
	j := j + 1;
	
END_FOR
END_METHOD

METHOD findSlot : BOOL
VAR_INPUT
	material : STRING;
END_VAR
VAR_OUTPUT
	index : INT := -1;
END_VAR
VAR
	i : DINT;
END_VAR
(*
IF materialID = '' THEN
	RETURN;
END_IF
*)
FOR i:=LOWER_BOUND(slots, 1) TO UPPER_BOUND(slots, 1) BY 1 DO
	IF slots[i].material = material THEN
		index := TO_INT(i);
		findSlot := TRUE;
		RETURN;
	END_IF
END_FOR
END_METHOD

METHOD getSlot : STRING
VAR_INPUT
	i : DINT;
END_VAR
VAR_OUTPUT
	occupancy : BOOL;
	error : BOOL;
END_VAR
error := i < LOWER_BOUND(slots, 1) OR i > UPPER_BOUND(slots, 1) (*OR slots = 0*);

IF error THEN
	RETURN;
END_IF

getSlot := slots[i].material;
occupancy := isOccupied(i := i, error => error);
END_METHOD

METHOD getSlotsAsArray : POINTER TO MaterialSlot
getSlotsAsArray := ADR(slots);
END_METHOD

METHOD isOccupied : BOOL
VAR_INPUT
	i : DINT;
END_VAR
VAR_OUTPUT
	error : BOOL;
END_VAR
error := i < LOWER_BOUND(slots, 1) OR i > UPPER_BOUND(slots, 1);

IF error THEN
	RETURN;
END_IF

isOccupied := slots[i].occupied;
END_METHOD

METHOD setSlot : BOOL
VAR_INPUT
	i : INT;
	material : STRING;
END_VAR
VAR_OUTPUT
	error : BOOL;
END_VAR
IF i < LOWER_BOUND(slots, 1) OR i > UPPER_BOUND(slots, 1) THEN
	error := TRUE;
	RETURN;
END_IF

slots[i].material := material;
END_METHOD

END_FUNCTION_BLOCK

// ---- DUTs/Containers/IntQueue.TcPOU
FUNCTION_BLOCK IntQueue EXTENDS Queue
VAR
	elements : FB_BA_DynamicArray := (uiEntrySize := SIZEOF(INT), uiMinExpCount := GVL.initArraySize);
	//length : USINT := 0;
END_VAR

METHOD clear : BOOL
VAR_INPUT
END_VAR
elements.Reset();
length := 0;
END_METHOD

METHOD contains : BOOL
VAR_INPUT
	value : INT;
END_VAR
VAR
	temp : INT;
	i : INT;
END_VAR
IF length = 0 THEN
	contains := FALSE;
	RETURN;
END_IF

FOR i:=0 TO (length-1) BY 1 DO
	temp := get(i);
	IF MEMCMP(ADR(temp), ADR(value), SIZEOF(INT)) = 0 THEN
		contains := TRUE;
		RETURN;
	END_IF
END_FOR
contains := FALSE;
END_METHOD

METHOD get : INT
VAR_INPUT
	i : INT;
END_VAR
elements.GetEntry(diIndex := i, pResultEntry := ADR(get));
END_METHOD

METHOD isEmpty : BOOL
VAR_INPUT
END_VAR
isEmpty := (elements.diCount = 0);
END_METHOD

METHOD poll : INT
VAR_INST
	temp : INT;
	i : UINT;
END_VAR
temp := get(i := 0);
elements.RemoveEntry(diIndex := 0);
//length := length - 1;
poll := temp;
END_METHOD

METHOD push : BOOL
VAR_INPUT
	value : INT;
END_VAR
elements.AddEntry(pEntry := ADR(value));
//length := length + 1;
END_METHOD

METHOD set : BOOL
VAR_INPUT
	i : INT;
	value : INT;
END_VAR
IF i > 0 AND i < length THEN
	elements.SetEntry(i, ADR(value));
	set := TRUE;
END_IF
END_METHOD

METHOD size : DINT
VAR_INPUT
END_VAR
size := elements.diCount;
END_METHOD

END_FUNCTION_BLOCK

// ---- DUTs/Containers/StringQueue.TcPOU
FUNCTION_BLOCK StringQueue EXTENDS Queue
VAR
	elements : FB_BA_DynamicArray := (uiEntrySize := SIZEOF(STRING), uiMinExpCount := GVL.initArraySize);
	//length : USINT := 0;
END_VAR

METHOD get : STRING
VAR_INPUT
	i : UINT;
END_VAR
elements.GetEntry(diIndex := i, pResultEntry := ADR(get));
END_METHOD

METHOD isEmpty : BOOL
VAR_INPUT
END_VAR
isEmpty := (elements.diCount = 0);
END_METHOD

METHOD poll : STRING
VAR_INST
	temp : STRING;
	i : UINT;
END_VAR
temp := get(i := 0);
elements.RemoveEntry(diIndex := 0);
//length := length - 1;
poll := temp;
END_METHOD

METHOD push : BOOL
VAR_INPUT
	value : STRING;
END_VAR
elements.AddEntry(pEntry := ADR(value));
//length := length + 1;
END_METHOD

METHOD size : DINT
VAR_INPUT
END_VAR
size := elements.diCount;
END_METHOD

END_FUNCTION_BLOCK

// ---- POUs/CallHardware.TcPOU
PROGRAM CallHardware

//conveyors
pushConveyorsToArray();
callConveyors();

//robots
robot1();
robot2();
robot3();
robot4();
//robot5();
//robot6();

//A23
wrapperA23();

//A22
skidA22Left();
skidA22Right();
magazineA22Left();
magazineA22Right();

insertionA22Left(
	enable:= TRUE, 
	slider:= verticalDriveA22Left, 
	screw:= horizontalDriveA22Left, 
	contact=> , 
	active=> , 
	error=> , 
	home=> , 
	homingComplete=> , 
	sliderPos=> );
	
insertionA22Right(
	enable:= TRUE, 
	slider:= verticalDriveA22Right, 
	screw:= horizontalDriveA22Right, 
	contact=> , 
	active=> , 
	error=> , 
	home=> , 
	homingComplete=> , 
	sliderPos=> );
	
pistonA22Bottom();
wrapperA22();

//A21
skidA21Left();
skidA21Right();

magazineA21Left();
magazineA21Right();

stagingTableLeft();
stagingTableRight();

strapperA21();

insertionA21Left(
	enable:= TRUE, 
	slider:= verticalDriveA21Left, 
	screw:= horizontalDriveA21Left, 
	contact=> , 
	active=> , 
	error=> , 
	home=> , 
	homingComplete=> , 
	sliderPos=> );
	
insertionA21Right(
	enable:= TRUE, 
	slider:= verticalDriveA21Right, 
	screw:= horizontalDriveA21Right, 
	contact=> , 
	active=> , 
	error=> , 
	home=> , 
	homingComplete=> , 
	sliderPos=> );
	
pistonA21Bottom();

METHOD PRIVATE callConveyors : BOOL
VAR
	i : DINT;
END_VAR
//rewrite this method, call every conveyor individually
//calling via loop will not call derived implementations
(*
FOR i:=1 TO numConveyors BY 1 DO
	conveyorsArr[i]^(
		bEnable:= , 
		enable=> , 
		direction=> , 
		pulse=> , 
		reset=> , 
		error=> , 
		sensorEntry=> , 
		sensorExit=> , 
		requestLifter=> , 
		lifterEnable=> , 
		lifterDirection=> , 
		lifterPulse=> , 
		lifterReset=> , 
		lifterError=> , 
		extended=> , 
		retracted=> , 
		position=> , 
		velocity=> );
END_FOR
*)
END_METHOD

METHOD PRIVATE pushConveyorsToArray : BOOL
conveyorsArr[1] := ADR(A24_SC_C01);
conveyorsArr[2] := ADR(A24_LRC_C02);
conveyorsArr[3] := ADR(A24_SC_C03);
conveyorsArr[4] := ADR(A24_LRC_C04);
conveyorsArr[5] := ADR(A24_SC_C05);
conveyorsArr[6] := ADR(A24_LRC_C06);
conveyorsArr[7] := ADR(A24_SC_C07);
conveyorsArr[8] := ADR(A24_LRC_C08);
conveyorsArr[9] := ADR(A24_SC_C09);
conveyorsArr[10] := ADR(A24_LRC_C10);
conveyorsArr[11] := ADR(A24_SC_C11);
conveyorsArr[12] := ADR(A24_LRC_C12);
conveyorsArr[13] := ADR(A24_SC_C13);

conveyorsArr[14] := ADR(A23_LSC_C14);

conveyorsArr[15] := ADR(A22_SC_C15);
conveyorsArr[16] := ADR(A22_LSC_C16);
conveyorsArr[17] := ADR(A22_LSC_C17);

conveyorsArr[18] := ADR(A21_SC_C18);
conveyorsArr[19] := ADR(A21_LSC_C19);
conveyorsArr[20] := ADR(A21_LSC_C20);
conveyorsArr[21] := ADR(A21_LSC_C21);

conveyorsArr[22] := ADR(A25_SC_C22);
conveyorsArr[23] := ADR(A25_LSC_C23);
conveyorsArr[24] := ADR(A25_SC_C24);
conveyorsArr[25] := ADR(A25_LSLCC_C25);
conveyorsArr[26] := ADR(A25_SC_C26);
conveyorsArr[27] := ADR(A25_LSLCC_C27);
conveyorsArr[28] := ADR(A25_SC_C28);
conveyorsArr[29] := ADR(A25_LSC_C29);
conveyorsArr[30] := ADR(A25_SC_C30);
conveyorsArr[31] := ADR(A25_SC_C31);
conveyorsArr[32] := ADR(A25_SC_C32);
conveyorsArr[33] := ADR(A25_SC_C33);
conveyorsArr[34] := ADR(A25_SC_C34);
conveyorsArr[35] := ADR(A25_SC_C35);
conveyorsArr[36] := ADR(A25_SC_C36);
conveyorsArr[37] := ADR(A25_SC_C37);
conveyorsArr[38] := ADR(A25_SC_C38);
END_METHOD

END_PROGRAM

// ---- POUs/ConveyorControlUnit.TcPOU
FUNCTION_BLOCK ConveyorControlUnit
VAR_IN_OUT
	conveyors : ARRAY[*] OF POINTER TO ConveyorSC;
END_VAR
VAR
	firstConveyor : DINT;
	lastConveyor : DINT;
	
	spoolTimer : TON;
	i : DINT := 1;
END_VAR
VAR CONSTANT
	spoolSpacing : TIME := T#100MS;
END_VAR

firstConveyor := LOWER_BOUND(conveyors, 1);
lastConveyor := UPPER_BOUND(conveyors, 1);

linkCompute();

spoolTimer(IN:= , PT:= spoolSpacing, Q=> , ET=> );
spoolTimer.IN := TRUE;
IF
	(conveyors[i]^.requestedMode = ConveyorMode.FORWARD OR conveyors[i]^.requestedMode = ConveyorMode.BACKWARD) AND //conveyor requests motion
	conveyors[i]^.requestedMode <> conveyors[i]^.trueMode AND //conveyor request differs from current operation
	spoolTimer.Q //ready to spool
THEN
	//spool up conveyor
	i := (i + 1) MOD (lastConveyor - firstConveyor + 1) + 1;
	spoolTimer.IN := FALSE;
END_IF

METHOD PRIVATE linkCompute : BOOL
VAR
	i : DINT;
	j : DINT;
	
	linkStart : DINT := -1;
	linkEnd : DINT := -1;
	
	priorityInLink : ConveyorMode;
END_VAR
(*
link interation method 
slower, but will correctly set all operations every cycle
*)
FOR i:=LOWER_BOUND(conveyors, 1) TO UPPER_BOUND(conveyors, 1) BY 1 DO
	IF conveyors[i]^.IsOccupied THEN
		
		IF linkStart = -1 THEN
			linkStart := i;
		END_IF
		
		priorityInLink := MAX(priorityInLink, conveyors[i]^.requestedMode);
		linkEnd := i;
		
	ELSIF linkStart <> -1 AND linkEnd <> -1 THEN //set all conveyor operations to priorityInLink
		linkEnd := i-1;
		
		FOR j:=linkStart TO linkEnd BY 1 DO
			conveyors[j]^.setMode(priorityInLink);
		END_FOR
		
		linkStart := -1;
		linkEnd := -1;
		priorityInLink := ConveyorMode.IDLE;
		
		CONTINUE;
	END_IF
	
END_FOR

IF linkStart > -1 AND linkEnd > -1 THEN
	FOR j:=linkStart TO linkEnd BY 1 DO
		conveyors[j]^.setMode(priorityInLink);
	END_FOR
END_IF
END_METHOD

END_FUNCTION_BLOCK

// ---- POUs/Helper Functions/Document/CreateJsonDocumentManual.TcPOU
FUNCTION CreateJsonDocumentManual : STRING(1000)
VAR_INPUT
	MaterialID : STRING;
	CheckFor : STRING;
	CameraNumber : INT;
END_VAR
VAR
	fbJson : FB_JsonSaxWriter;
END_VAR

fbJson.StartObject();

fbJson.AddKey('MaterialID');
fbJson.AddString(MaterialID);

fbJson.AddKey('CheckFor');
fbJson.AddString(CheckFor);

fbJson.AddKey('CameraNumber');
fbJson.AddString(CameraNumber);

//below are keys for VisionPC to write to
fbJson.AddKey('SuccessFlag');
fbJson.AddKey('OrientAdjustX');
fbJson.AddKey('OrientAdjustY');
fbJson.AddKey('OrientAdjustX');

fbJson.EndObject();

CreateJsonDocumentManual := fbJson.GetDocument();

END_FUNCTION

// ---- POUs/Helper Functions/General/BundleIsValid.TcPOU
FUNCTION BundleIsValid : BOOL
VAR_INPUT
	b : REFERENCE TO Bundle;
END_VAR

BundleIsValid := NOT(b.id = '');

END_FUNCTION

// ---- POUs/Helper Functions/General/PositionIsValid.TcPOU
FUNCTION PositionIsValid : BOOL
VAR_INPUT
	pair : REFERENCE TO PositionMaterials;
END_VAR

PositionIsValid := (
	pair.position <> -1 AND
	(
		pair.top <> '' OR
		pair.left <> '' OR
		pair.right <> '' OR
		pair.bottom <> '' OR
		
		pair.topLeft <> '' OR
		pair.topRight <> '' OR
		pair.bottomLeft <> '' OR
		pair.bottomRight <> ''
	));

END_FUNCTION

// ---- POUs/Helper Functions/Hardware Modules/SetupHardware.TcPOU
FUNCTION SetupHardware : BOOL
VAR
	iWoodBunkSlot : WoodBunk;
	iChipboardSlot : Chipboard;
	
	i : INT;
END_VAR

FOR iWoodBunkSlot:=1 TO WoodBunk.size-1 BY 1 DO //init wood bunk magazine slots
	magazineA21Left.setSlot(i := iWoodBunkSlot, material := TO_STRING(iWoodBunkSlot), error => );
	magazineA21Right.setSlot(i := iWoodBunkSlot, material := TO_STRING(iWoodBunkSlot), error => );
END_FOR

//--------------------------------------------------

FOR iChipboardSlot:=1 TO Chipboard.size-1 BY 1 DO //init chipboard skid slots
	skidA21Left.setSlot(i := iChipboardSlot, material := TO_STRING(iChipboardSlot), error => );
	skidA21Right.setSlot(i := iChipboardSlot, material := TO_STRING(iChipboardSlot), error => );
END_FOR

//--------------------------------------------------

FOR i:=1 TO GVL.maxQueue BY 1 DO //get wood bunk magazine + chipboard skid availability from robot1 and robot2
	{warning disable C0195}
	skidA21Left.setOccupancy( i := i, occupancy := IntegerBitAccess(robot1.inputs[4], i-1) );
	skidA21Right.setOccupancy( i := i, occupancy := IntegerBitAccess(robot2.inputs[4], i-1) );

	magazineA21Left.setOccupancy( i := i, occupancy := IntegerBitAccess(robot1.inputs[3], i-1) );
	magazineA21Right.setOccupancy( i := i, occupancy := IntegerBitAccess(robot2.inputs[3], i-1) );
END_FOR

//--------------------------------------------------

//enable all drives
verticalDriveA21Left.bEnable := TRUE;
verticalDriveA21Right.bEnable := TRUE;
insertionA21Left.enable := TRUE;
horizontalDriveA21Left.bEnable := TRUE;
horizontalDriveA21Right.bEnable := TRUE;
insertionA21Right.enable := TRUE;
pistonA21Bottom.bEnable := TRUE;

SetupHardware := TRUE;

END_FUNCTION

// ---- POUs/Helper Functions/Utility/IntegerBitAccess.TcPOU
FUNCTION IntegerBitAccess : BOOL
VAR_INPUT
	num : ULINT;
	n : ULINT;
END_VAR

IntegerBitAccess := (SHR(num, n) AND 1) > 0;

END_FUNCTION

// ---- POUs/Helper Functions/Utility/CleanStringsArray.TcPOU
FUNCTION CleanStringsArray : BOOL
VAR_IN_OUT
	arr : ARRAY[*] OF STRING;
END_VAR
VAR
	i : DINT;
END_VAR

FOR i:=LOWER_BOUND(arr, 1) TO UPPER_BOUND(arr, 1) BY 1 DO
	IF arr[i] = '' THEN
		MEMSET(ADR(arr[i]), 0, SIZEOF(arr[i]));
	END_IF
END_FOR

END_FUNCTION

// ---- POUs/Helper Functions/Utility/WithinTolerance.TcPOU
FUNCTION WithinTolerance : BOOL
VAR_INPUT
	v1 : LREAL;
	v2 : LREAL;
	tolerance : LREAL;
END_VAR
(*
checks if v1 close enough to v2 within a given margin
*)

WithinTolerance := ABS(v1-v2) < tolerance;

END_FUNCTION

// ---- POUs/MAIN.TcPOU
PROGRAM MAIN
VAR_OUTPUT //globally readable, but only modifiable by MAIN
	outputBuffer : ARRAY[Surface.LEFT..Surface.RIGHT] OF Bundle;
	outputBufferPass, outputBufferFail : Bundle;
	numOutputBundles : USINT := 0;
	
	bundleIn : Bundle;
	bundleOut : Bundle;
	
	start : BOOL;
	
	ready : BOOL;
	busy : BOOL;
	done : BOOL;
	error : BOOL;
	backlog : BOOL;
	
	stop : BOOL;
	execute : BOOL;
	hold : BOOL;
	reset : BOOL;
	
	localTime : TIMESTRUCT;
	
	pmlModeString : STRING;
	pmlStateString : STRING;
END_VAR
VAR
	clearPassBuffer, clearFailBuffer AT %I* : BOOL;
	receiverStruct : AdsData;
	
	//ETA is not strictly required, area will process bundle even if it is not in ETA arrays
	expectedBundles : ARRAY[0..GVL.maxQueue] OF STRING; //bundles expected to arrive
	expectedArrivals : ARRAY[0..GVL.maxQueue] OF TIMESTRUCT; //bundles expected to arrive
	numEtaBundles : INT;
	
	//parallel arrays - bundle, bypass
	numBundles : INT;
	bundlesQueue : ARRAY[0..GVL.maxQueue] OF Bundle;
	bundlesBypass : ARRAY[0..GVL.maxQueue] OF BOOL;
END_VAR
VAR
	//spacerRecollector : PackagerFreeAsync;
	//paperSection : PaperEx;
	//cardboardCornerGuardSection : CardboardCornerGuardEx;
	//chipboardSection : ChipboardEx;
	woodBunkSection : WoodBunkEx;
	//outputSection : AreaOutputEx;	
END_VAR
VAR
	fbLocalSystemTime : FB_LocalSystemTime;
	dbLogger : SqlDatabaseAccessor;
	conveyorController : ConveyorControlUnit;
	
	pmlState : E_PMLState;
	pmlCommand : E_PMLCommand;
	pmlStateMachine : PML_StateMachine;
	
	pmlModeRequest : E_PMLCustomUnitMode := ePMLCustomUnitMode_Production;
	pmlMode : E_PMLCustomUnitMode;
	pmlModeManager : PML_UnitModeManager;
END_VAR
VAR //these variables are only tracked for HMI
	sectionsBusy : ARRAY[0..SectionEnum.size] OF BOOL;
	sectionsIterator : ARRAY[0..SectionEnum.size] OF INT;
END_VAR

(*
ready := paperSection.ready; //if A2 is not ready, dispatch controller must block operator from sending bundles here
busy := paperSection.busy OR cardboardCornerGuardSection.busy OR chipboardSection.busy OR woodBunkSection.busy OR outputSection.busy;
done := outputSection.done;
backlog := numBundlesQueue > 5;
*)

CallHardware(); //start program with CallHardware()
SetupHardware(); //set bEnables, setup material holder slots, etc

initialize();

fillBundlesQueue();

SizeCheck();
getLocalTime();

AdsClient( //PLC-PLC comms
	ServerNetId:= , 
	ServerPort:= , 
	bBusy=> , 
	err=> , 
	errid=> , 
	localPrgName=> , 
	localNetId=> , 
	localPort=> , 
	socketReady=> , 
	remoteAccessPrefix=> );
	
TcpServer1Vision( //PLC-Vision comms
	ServerNetId:= , 
	ServerAdr:= , 
	ServerPort:= , 
	busy=> , 
	error=> , 
	errorId=> , 
	bytesReceived=> , 
	connected=> , 
	receiveStruct=> );
	
runPML();

IF AdsClient.fetchData(receiverStruct) THEN
	interpretTransmission(receiverStruct);
END_IF


IF ready AND BundleIsValid(bundleIn) THEN
	receive();
END_IF


IF clearPassBuffer OR clearFailBuffer THEN
	transfer();
	shiftBundles();
END_IF

dbLogger();

conveyorController(conveyors := conveyorsArr);
CallHardware(); //start program with CallHardware()

METHOD fillBundlesQueue : BOOL
VAR
	i : INT;
END_VAR
IF NOT start THEN //for HMI testing only, remove for production
	FOR i:=0 TO GVL.maxQueue BY 1 DO
		bundlesQueue[i].id := TO_STRING(i);
	END_FOR
	
	start := TRUE;
END_IF
END_METHOD

METHOD PRIVATE getLocalTime : BOOL
fbLocalSystemTime(
	sNetID:= '', 
	bEnable:= TRUE, 
	dwCycle:= , 
	dwOpt:= , 
	tTimeout:= , 
	bValid=> , 
	systemTime=> localTime, 
	tzID=> );
	
getLocalTime := TRUE;
END_METHOD

METHOD PRIVATE initialize : BOOL
//paperSection.connectTo(ADR(cardboardCornerGuardSection));
//cardboardCornerGuardSection.connectTo(ADR(chipboardSection));
//chipboardSection.connectTo(ADR(woodBunkSection));
woodBunkSection.connectTo(0); //(ADR(outputSection));
//connecting to 0 means no next section

//paperSection.sectionID := SectionEnum.PAPER;
//cardboardCornerGuardSection.sectionID := SectionEnum.CARDBOARD_CORNERGUARD;
//chipboardSection.sectionID := SectionEnum.CHIPBOARD;
woodBunkSection.sectionID := SectionEnum.WOOD_BUNK;
//outputSection.sectionID := SectionEnum.OUTPUT;

(*
	paperSection.pNextSection := ADR(cardboardCornerGuardSection);
	cardboardCornerGuardSection.accessNextSection := ADR(chipboardSection);
	chipboardSection.accessNextSection := ADR(woodBunkSection);
	woodBunkSection.accessNextSection := ADR(outputSection);
	outputSection.accessNextSection := 0;
*)

initialize := TRUE;
END_METHOD

METHOD PRIVATE interpretTransmission : BOOL
VAR_INPUT
	data : REFERENCE TO AdsData;
END_VAR
VAR
	i : INT;
END_VAR
CASE data.description OF
	EventsEnum.BUNDLE_IN:
		MEMCPY(ADR(bundleIn), ADR(data.binaryData), SIZEOF(bundleIn));
			
	EventsEnum.BUNDLE_ETA:
		MEMCPY(ADR(expectedBundles[numEtaBundles]), ADR(data.binaryData), SIZEOF(expectedBundles[numEtaBundles]));
		expectedArrivals[numEtaBundles] := data.timestamp;
		
END_CASE
END_METHOD

METHOD maintenance : BOOL
VAR_INPUT
END_VAR
END_METHOD

METHOD PRIVATE process : BOOL
(*
full parallel processsing
all sections may operate concurrently on any bundle
*)
(*
paperSection(
	enable:= run[SectionEnum.PAPER], 
	bundlesQueue:= bundlesQueue, 
	bundlesBypass:= bundlesBypass,
	bundleOut=> , 
	bypass=> , 
	ready=> , 
	busy=> sectionsBusy[SectionEnum.PAPER], 
	done=> , 
	error=> , 
	backlog=> ,
	iBundle=> sectionsIterator[SectionEnum.PAPER],
	iPair=> );
	
cardboardCornerGuardSection(
	enable:= run[SectionEnum.CARDBOARD_CORNERGUARD],
	bundlesQueue:= bundlesQueue, 
	bundlesBypass:= bundlesBypass,
	bundleOut=> ,
	bypass=> , 
	ready=> , 
	busy=> sectionsBusy[SectionEnum.CARDBOARD_CORNERGUARD], 
	done=> , 
	error=> , 
	backlog=> ,
	iBundle=> sectionsIterator[SectionEnum.CARDBOARD_CORNERGUARD],
	iPair=> );

chipboardSection(
	enable:= run[SectionEnum.CHIPBOARD],
	bundlesQueue:= bundlesQueue, 
	bundlesBypass:= bundlesBypass, 
	bundleOut=> ,
	bypass=> , 
	ready=> , 
	busy=> sectionsBusy[SectionEnum.CHIPBOARD], 
	done=> , 
	error=> , 
	backlog=> ,
	iBundle=> sectionsIterator[SectionEnum.CHIPBOARD],
	iPair=> );
*)

(*
woodBunkSection(
	enable:= run[SectionEnum.WOOD_BUNK],
	bundlesQueue:= bundlesQueue, 
	bundlesBypass:= bundlesBypass, 
	bundleOut=> ,
	bypass=> , 
	ready=> , 
	busy=> sectionsBusy[SectionEnum.WOOD_BUNK], 
	done=> , 
	error=> , 
	backlog=> ,
	iBundle=> sectionsIterator[SectionEnum.WOOD_BUNK],
	iPair=> );
*)
(*
outputSection(
	enable:= run[SectionEnum.OUTPUT],
	bundlesQueue:= bundlesQueue, 
	bundlesBypass:= bundlesBypass,
	outputBuffer:= outputBuffer,
	bundleOut=> , 
	bypass=> , 
	ready=> , 
	busy=> sectionsBusy[SectionEnum.OUTPUT],
	done=> , 
	error=> , 
	backlog=> ,
	iBundle=> sectionsIterator[SectionEnum.OUTPUT],
	iPair=> );
*)
END_METHOD

METHOD PRIVATE processLLD : BOOL
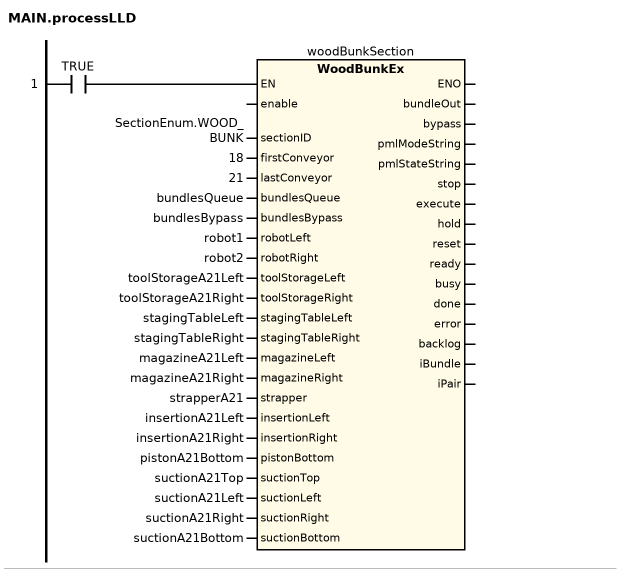
// NETWORK 1
woodBunkSection(
    sectionID := SectionEnum.WOOD_BUNK,
    firstConveyor := 18,
    lastConveyor := 21,
    bundlesQueue := bundlesQueue,
    bundlesBypass := bundlesBypass,
    robotLeft := robot1,
    robotRight := robot2,
    toolStorageLeft := toolStorageA21Left,
    toolStorageRight := toolStorageA21Right,
    stagingTableLeft := stagingTableLeft,
    stagingTableRight := stagingTableRight,
    magazineLeft := magazineA21Left,
    magazineRight := magazineA21Right,
    strapper := strapperA21,
    insertionLeft := insertionA21Left,
    insertionRight := insertionA21Right,
    pistonBottom := pistonA21Bottom,
    suctionTop := suctionA21Top,
    suctionLeft := suctionA21Left,
    suctionRight := suctionA21Right,
    suctionBottom := suctionA21Bottom); // WoodBunkEx
END_METHOD

METHOD PRIVATE ps_AbortCondition : BOOL
VAR_INPUT
END_VAR
END_METHOD

METHOD PRIVATE ps_Aborted : BOOL
VAR_INPUT
END_VAR
END_METHOD

METHOD PRIVATE ps_Aborting : BOOL
VAR_INPUT
END_VAR
END_METHOD

METHOD PRIVATE ps_Clearing : BOOL
VAR_INPUT
END_VAR
END_METHOD

METHOD PRIVATE ps_Complete : BOOL
VAR_INPUT
END_VAR
END_METHOD

METHOD PRIVATE ps_Completing : BOOL
VAR_INPUT
END_VAR
END_METHOD

METHOD PRIVATE ps_Execute : BOOL
VAR_INPUT
END_VAR
VAR_OUTPUT
	error : BOOL;
END_VAR
CASE pmlMode OF
	0: //invalid mode
	ePMLCustomUnitMode_Production:		ps_Execute := process();
	ePMLCustomUnitMode_Maintenance:		maintenance();
	ePMLCustomUnitMode_Manual:			//
	ePMLCustomUnitMode_SemiAuto:		ps_Execute := process(); //manually step bundle into area - sections may be auto while area is semi-auto
END_CASE
END_METHOD

METHOD PRIVATE ps_Held : BOOL
VAR_INPUT
END_VAR
END_METHOD

METHOD PRIVATE ps_HoldCondition : BOOL
VAR_INPUT
END_VAR
END_METHOD

METHOD PRIVATE ps_Holding : BOOL
VAR_INPUT
END_VAR
END_METHOD

METHOD PRIVATE ps_Idle : BOOL
VAR_INPUT
END_VAR
(*
IF BundleIsValid(currentBundle) THEN
	ps_Idle := TRUE;
	done := FALSE;
END_IF
*)

ps_Idle := TRUE; (*start section input*)
END_METHOD

METHOD PRIVATE ps_Resetting : BOOL
VAR_INPUT
END_VAR
END_METHOD

METHOD PRIVATE ps_Starting : BOOL
VAR_INPUT
END_VAR
END_METHOD

METHOD PRIVATE ps_StopCondition : BOOL
VAR_INPUT
END_VAR
END_METHOD

METHOD PRIVATE ps_Stopped : BOOL
VAR_INPUT
END_VAR
END_METHOD

METHOD PRIVATE ps_Stopping : BOOL
VAR_INPUT
END_VAR
END_METHOD

METHOD PRIVATE ps_SuspendCondition : BOOL
VAR_INPUT
END_VAR
END_METHOD

METHOD PRIVATE ps_Suspended : BOOL
VAR_INPUT
END_VAR
END_METHOD

METHOD PRIVATE ps_Suspending : BOOL
VAR_INPUT
END_VAR
END_METHOD

METHOD PRIVATE ps_Unholding : BOOL
VAR_INPUT
END_VAR
END_METHOD

METHOD PRIVATE ps_Unsuspending : BOOL
VAR_INPUT
END_VAR
END_METHOD

{attribute 'TcRpcEnable'}
METHOD PRIVATE receive : BOOL
VAR
	i : INT;
	shiftIndex : INT := -1;
	invalidBundle : Bundle;
END_VAR
FOR i:=0 TO GVL.maxQueue BY 1 DO //find the bundle in the ETA queue
	IF expectedBundles[i] = bundleIn.id THEN
		shiftIndex := i;
		EXIT;
	END_IF
END_FOR

IF shiftIndex > -1 THEN //if the bundle is found in the ETA queue, shift everything down
	MEMMOVE(
		ADR(expectedBundles[shiftIndex]), 
		ADR(expectedBundles[shiftIndex + 1]), 
		SIZEOF(STRING) * TO_UINT(GVL.maxQueue - shiftIndex));
		
	MEMMOVE(
		ADR(expectedArrivals[shiftIndex]), 
		ADR(expectedArrivals[shiftIndex + 1]), 
		SIZEOF(TIMESTRUCT) * TO_UINT(GVL.maxQueue - shiftIndex) );
		
	numEtaBundles := numEtaBundles - 1;
END_IF

FOR i:=0 TO GVL.maxQueue BY 1 DO
	IF BundleIsValid(bundlesQueue[i]) AND NOT bundlesBypass[i] THEN
		bundlesQueue[i] := bundleIn;
		bundlesBypass[i] := FALSE;
		
		receive := TRUE;
		RETURN;
	END_IF
END_FOR

IF NOT receive THEN
	error := TRUE;
END_IF
END_METHOD

METHOD PRIVATE runPML : BOOL
(*
PackML
	state machine for packaging applications - see Tc3_PackML_V2 library on InfoSys
	
	final states - wait for an input or condition and command to new state
	intermediate states - complete a task and call pmlStateMachine.M_StateComplete() to advance to next state
	
the following states currently use the same logic (albeit in different methods), implementation may change later
	ps_Stopping() and ps_Aborting()
	ps_Resetting() and ps_Clearing()
	
STOP - controlled stop **with intent to shutdown or vacate for extended time** induced by operator/HMI - otherwise use HOLD
ABORT - emergency stop due to machine errors


HOLD - minor local issues
SUSPEND - external issues

EXECUTE - major control logic
	different modes may require different tasks
	create methods as required for different modes, then call the correct method in ps_Completing()
	can be commanded to STOP, ABORT, HOLD, or SUSPEND at any point
COMPLETING - process complete, move product out of system and finish transition to COMPLETED

the implementation below can be copied to all POUs that use a PackML state machine
the individual ps_< > methods need to be implemented for the specific application
*)
IF ps_AbortCondition() THEN //abort condition
	pmlCommand := ePMLCommand_Abort;
ELSIF ps_StopCondition() THEN //stop condition
	pmlCommand := ePMLCommand_Stop;
END_IF

CASE pmlState OF
	0 (*ePMLState_Undefined*): //default state on startup
		pmlCommand := ePMLCommand_Stop;
		
	ePMLState_Stopping:
		IF ps_Stopping() THEN
			pmlStateMachine.M_StateComplete();
		END_IF
		
	ePMLState_Stopped:
		IF ps_Stopped() THEN
			pmlCommand := ePMLCommand_Reset;
		END_IF
	
    ePMLState_Resetting:
		IF ps_Resetting() THEN
			pmlStateMachine.M_StateComplete();
		END_IF
		
	ePMLState_Idle:
		IF ps_Idle() THEN
			pmlCommand := ePMLCommand_Start;
		END_IF		
	
	ePMLState_Starting:
		IF ps_Starting() THEN
			pmlStateMachine.M_StateComplete();
		END_IF
	
	ePMLState_Execute: //check the conditions in order of their priority, currently HOLD has the highest priority
		IF ps_HoldCondition() THEN
			pmlCommand := ePMLCommand_Hold;
			
		ELSIF ps_SuspendCondition() THEN
			pmlCommand := ePMLCommand_Suspend;			
		
		ELSIF ps_Execute(error => error) THEN //ps_Execute.error => THIS^.error
			pmlStateMachine.M_StateComplete();
			pmlCommand := ePMLCommand_Complete;
		END_IF
		
	ePMLState_Completing:
		IF ps_Completing() THEN
			pmlStateMachine.M_StateComplete();
		END_IF
	
	ePMLState_Complete:
		IF ps_Complete() THEN
			pmlCommand := ePMLCommand_Reset;
		END_IF
	
	ePMLState_Holding:
		IF ps_Holding() THEN
			pmlStateMachine.M_StateComplete();
		END_IF
	
	ePMLState_Held:
		IF NOT hold THEN
			pmlCommand := ePMLCommand_Unhold;
		END_IF
	
	ePMLState_Unholding:
		IF ps_Unholding() THEN
			pmlStateMachine.M_StateComplete(); //release all pause commands and IO
		END_IF
		
	ePMLState_Suspending: //based on next section conditions
		IF ps_Suspending() THEN
			pmlStateMachine.M_StateComplete();
		END_IF
		
	ePMLState_Suspended: //based on next section conditions
		IF ps_Suspended() THEN
			pmlCommand := ePMLCommand_Unsuspend;
		END_IF
	
	ePMLState_Unsuspending: //based on next section conditions
		IF ps_Unsuspending() THEN
			pmlStateMachine.M_StateComplete();
		END_IF
	
	ePMLState_Aborting:
		IF ps_Aborting() THEN
			pmlStateMachine.M_StateComplete();
		END_IF
	
	ePMLState_Aborted:
		IF ps_Aborted() THEN
			pmlCommand := ePMLCommand_Clear;
		END_IF
	
	ePMLState_Clearing:
		IF ps_Clearing() THEN
			pmlStateMachine.M_StateComplete();
		END_IF
	
END_CASE
END_METHOD

METHOD shiftBundles : BOOL
VAR_INPUT
END_VAR
//shift down parallel arrays
MEMMOVE(ADR(bundlesQueue[0]), ADR(bundlesQueue[1]), SIZEOF(Bundle) * TO_UINT(GVL.maxQueue));
MEMMOVE(ADR(bundlesBypass[0]), ADR(bundlesBypass[1]), SIZEOF(BOOL) * TO_UINT(GVL.maxQueue));

//decrement each section's iterator to realign with their correct bundle
//paperSection.shiftIterator();
//cardboardCornerGuardSection.shiftIterator();
//chipboardSection.shiftIterator();
woodBunkSection.shiftIterator();
//outputSection.shiftIterator();
END_METHOD

METHOD PRIVATE transfer : BOOL
VAR
	i : INT;
END_VAR
//send TCP/ADS transmission back to Dispatch once bundle is removed from the plant

IF clearPassBuffer THEN
	dbLogger.queueEvent(event:= EventsEnum.BUNDLE_OUT); //modify to include bundle ID
	//outputBufferPass := GVL.nullBundle;
	MEMSET(ADR(outputBufferPass), 0, SIZEOF(outputBufferPass));
END_IF

IF clearFailBuffer THEN
	dbLogger.queueEvent(event:= EventsEnum.BUNDLE_OUT); //modify to include bundle ID
	//outputBufferFail := GVL.nullBundle;
	MEMSET(ADR(outputBufferFail), 0, SIZEOF(outputBufferFail));
END_IF
END_METHOD

END_PROGRAM

// ---- Sections/A21b - Wood Bunk/WoodBunkEx.TcPOU
FUNCTION_BLOCK WoodBunkEx EXTENDS SectionEx
VAR_IN_OUT //references to required hardware
	robotLeft, robotRight : RobotA21;
	toolStorageLeft, toolStorageRight : A21ToolStorage;
	
	stagingTableLeft, stagingTableRight : StagingTable;
	magazineLeft, magazineRight : SkidMagazine;
	
	strapper : StrapMachine;
	
	insertionLeft, insertionRight : Insertion;
	pistonBottom : SimplePiston;
	
	suctionTop : ARRAY[*] OF SuctionPad; (*1..3*)
	suctionLeft : ARRAY[*] OF SuctionPad; (*1..4*)
	suctionRight : ARRAY[*] OF SuctionPad; (*1..4*)
	suctionBottom : ARRAY[*] OF SuctionPad; (*1..2*)
END_VAR
VAR
	conveyorPos : REAL;
	
	step : (IDLE, STAGING, LOAD_WB, PUSH, STRAP, RELEASE, COMPLETE := 1050);
	
	stageStepLeft, stageStepRight : INT;
	loadStepLeft, loadStepRight : INT;
END_VAR
VAR //bundle data
	demoHeight : REAL := 640; //mm
	materialsArr : (*REFERENCE TO*) ARRAY[0..GVL.maxPairs] OF PositionMaterials;
END_VAR
VAR
	//AOIs encapsulate functionality and reduce the number of module variables
	aoiTemplateLeft, aoiTemplateRight : AOI_StagingTemplate;
	aoiStageLeft, aoiStageRight : AOI_StageWoodBunk; 
	aoiLoadLeft, aoiLoadRight : AOI_LoadWoodBunk;
	
	suctionRelease : TON;
	
	//for testing, to be removed when deployoed
	latchLeft, latchRight : BOOL; //prevents SMC sliders from overshooting
	suctionEnableTop, suctionEnableLeft, suctionEnableRight, suctionEnableBottom : BOOL;
END_VAR

blocks(); //call AOIs and large library FBs

SUPER^();

CASE status OF //add additional instructions for each state
	SectionTask.IDLE:
		//RETURN;
	
	SectionTask.ALIGNING:
		stage(error => error);
		
	SectionTask.ACTIVE:
		//
		
	SectionTask.CLEARING:
		aoiLoadLeft.reset();
		aoiLoadRight.reset();
		
		aoiStageLeft.reset();
		aoiStageRight.reset();
		
		aoiTemplateLeft.reset();
		aoiTemplateRight.reset();
		
	SectionTask.COMPLETE:	
		//
		
	-100:
		RETURN;
		
END_CASE

METHOD PROTECTED blocks : BOOL
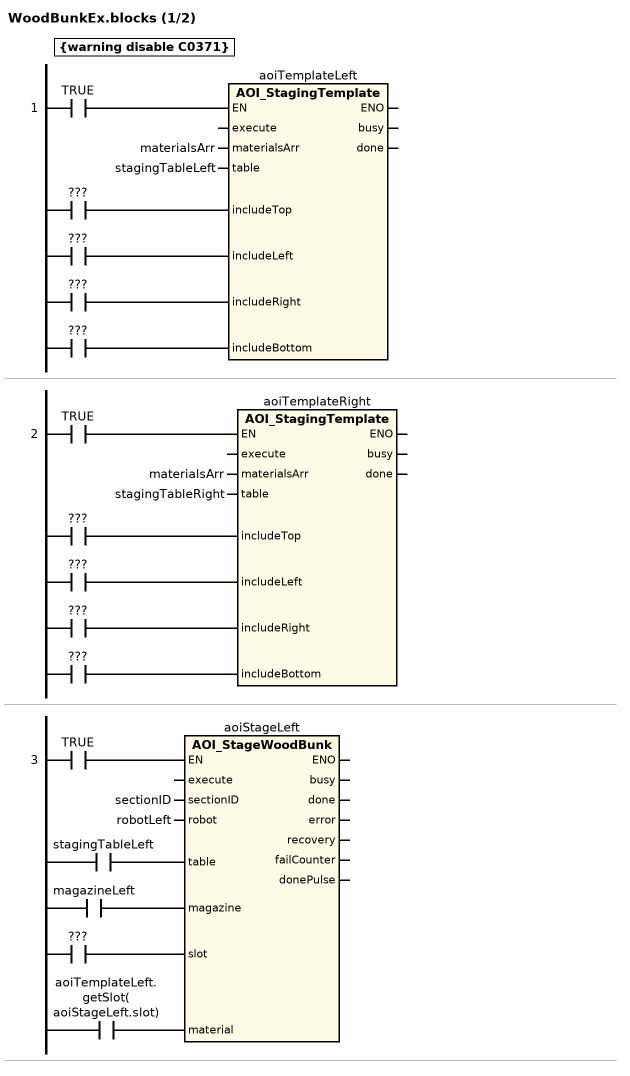
// NETWORK 1
// label: {warning disable C0371}
aoiTemplateLeft(materialsArr := materialsArr, table := stagingTableLeft); // AOI_StagingTemplate

// NETWORK 2
aoiTemplateRight(materialsArr := materialsArr, table := stagingTableRight); // AOI_StagingTemplate

// NETWORK 3
aoiStageLeft(
    sectionID := sectionID,
    robot := robotLeft,
    table := stagingTableLeft,
    magazine := magazineLeft,
    material := aoiTemplateLeft.getSlot(aoiStageLeft.slot)); // AOI_StageWoodBunk

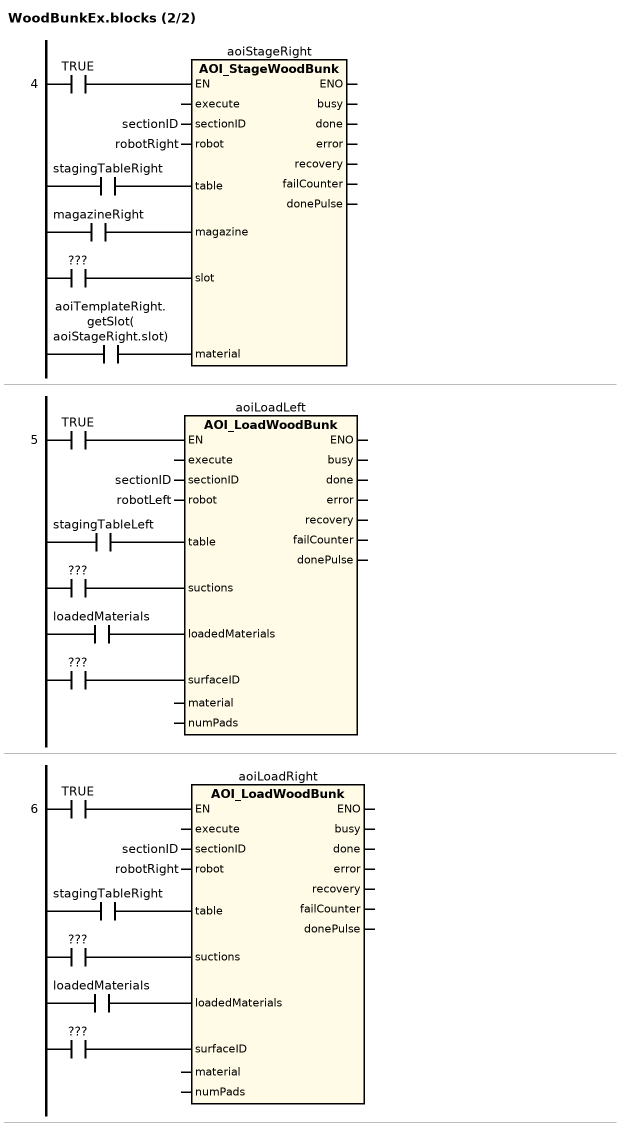
// NETWORK 4
aoiStageRight(
    sectionID := sectionID,
    robot := robotRight,
    table := stagingTableRight,
    magazine := magazineRight,
    material := aoiTemplateRight.getSlot(aoiStageRight.slot)); // AOI_StageWoodBunk

// NETWORK 5
aoiLoadLeft(
    sectionID := sectionID,
    robot := robotLeft,
    table := stagingTableLeft,
    loadedMaterials := loadedMaterials); // AOI_LoadWoodBunk

// NETWORK 6
aoiLoadRight(
    sectionID := sectionID,
    robot := robotRight,
    table := stagingTableRight,
    loadedMaterials := loadedMaterials); // AOI_LoadWoodBunk
END_METHOD

METHOD PROTECTED callLocalModules : BOOL
VAR_INPUT
END_VAR
{warning disable C0371}
(*
insertionLeft(
	enable:= TRUE, 
	slider:= verticalDriveLeft, 
	screw:= horizontalDriveLeft, 
	contact=> , 
	softContact=> , 
	active=> , 
	error=> , 
	home=> , 
	homingComplete=> , 
	sliderPos=> );
	
insertionRight(
	enable:= TRUE, 
	slider:= verticalDriveRight, 
	screw:= horizontalDriveRight,  
	contact=> , 
	softContact=> , 
	active=> , 
	error=> , 
	home=> , 
	homingComplete=> , 
	sliderPos=> );
*)
suctionRelease(IN:= , PT:= suctionReleaseDelay, Q=> , ET=> );
END_METHOD

METHOD PROTECTED discharge : BOOL
VAR_INPUT
END_VAR
//unload from insertion
//remove from staging table
END_METHOD

METHOD PROTECTED load : BOOL
VAR_INPUT
	pairIndex : INT;
END_VAR
VAR_OUTPUT
	error : BOOL;
END_VAR
VAR
	pair : REFERENCE TO PositionMaterials REF= materialsArr[pairIndex];
	errorLeft, errorRight : BOOL;
END_VAR
{warning disable C0371}
(*
this is the new code for loading wood bunks from staging table to insertion
loading sequences are independent as each side has its own step variable
can be extended by changing the include<> parameters
*)

load :=
	loadEx(
		robot:= robotLeft, 
		aoiLoad:= aoiLoadLeft, 
		loadStep:= loadStepLeft, 
		pairIndex:= pairIndex, 
		includeTop:= TRUE, 
		includeLeft:= TRUE, 
		includeRight:= FALSE, 
		includeBottom:= FALSE, 
		error=> errorLeft)
	AND
	loadEx(
		robot:= robotRight, 
		aoiLoad:= aoiLoadRight, 
		loadStep:= loadStepRight, 
		pairIndex:= pairIndex, 
		includeTop:= FALSE, 
		includeLeft:= FALSE, 
		includeRight:= TRUE, 
		includeBottom:= TRUE, 
		error=> errorRight);
		
error := errorLeft OR errorRight;

(*
below is the old code for loading wood bunks from staging table to insertion
it loads wood bunks in sets - top/bottom, then sides
if one side is finished loading a set before the other, it waits until the other side is done before advancing the set
*)
(*
IF robotLeft.error OR robotRight.error THEN
	error := TRUE;
	RETURN;
	
ELSIF 
	(robotLeft.reservation <> sectionID AND_THEN NOT robotLeft.reserve(sectionID)) OR 
	(robotRight.reservation <> sectionID AND_THEN NOT robotRight.reserve(sectionID))
THEN //loading requires both robots be reserved together
	RETURN;
	
ELSIF //robots have wrong tool
	(robotLeft.tool <> sectionID AND_THEN NOT robotLeft.changeEOAT(targetTool := sectionID)) OR
	(robotRight.tool <> sectionID AND_THEN NOT robotRight.changeEOAT(targetTool := sectionID))
THEN
	RETURN;
	
END_IF

CASE loadStep OF
	0: //top and bottom
		IF aoiLoadLeft.done AND aoiLoadRight.done THEN
			aoiLoadLeft.execute := aoiLoadRight.execute := FALSE;
			aoiLoadLeft.material := aoiLoadRight.material := '';
			
			aoiLoadLeft.reset();
			aoiLoadRight.reset();
			loadStep := 10;
			RETURN;
		END_IF
		
		aoiLoadLeft.suctions := suctionTop;
		aoiLoadLeft.surfaceID := Surface.TOP;
		aoiLoadLeft.material := pair.top;
		aoiLoadLeft.numPads := UPPER_BOUND(suctionTop, 1) - LOWER_BOUND(suctionTop, 1) + 1;
		
		aoiLoadRight.suctions := suctionBottom;
		aoiLoadRight.surfaceID := Surface.BOTTOM;
		aoiLoadRight.material := pair.bottom;
		aoiLoadRight.numPads := UPPER_BOUND(suctionBottom, 1) - LOWER_BOUND(suctionBottom, 1) + 1;
		
		aoiLoadLeft.execute := NOT aoiLoadLeft.done AND NOT aoiLoadLeft.busy;
		aoiLoadRight.execute := NOT aoiLoadRight.done AND NOT aoiLoadRight.busy;
		
	10: //sides
		IF aoiLoadLeft.done AND aoiLoadRight.done THEN
			aoiLoadLeft.execute := aoiLoadRight.execute := FALSE;
			aoiLoadLeft.material := aoiLoadRight.material := '';
			
			aoiLoadLeft.reset();
			aoiLoadRight.reset();
			loadStep := COMPLETE;
			RETURN;
		END_IF
		
		aoiLoadLeft.suctions := suctionLeft;
		aoiLoadLeft.surfaceID := Surface.LEFT;
		aoiLoadLeft.material := pair.left;
		aoiLoadLeft.numPads := UPPER_BOUND(suctionLeft, 1) - LOWER_BOUND(suctionLeft, 1) + 1;
		
		aoiLoadRight.suctions := suctionRight;
		aoiLoadRight.surfaceID := Surface.RIGHT;
		aoiLoadRight.material := pair.right;
		aoiLoadRight.numPads := UPPER_BOUND(suctionRight, 1) - LOWER_BOUND(suctionRight, 1) + 1;
		
		aoiLoadLeft.execute := NOT aoiLoadLeft.done AND NOT aoiLoadLeft.busy;
		aoiLoadRight.execute := NOT aoiLoadRight.done AND NOT aoiLoadRight.busy;
		
	COMPLETE:				
		robotLeft.release(sectionID);
		robotRight.release(sectionID);
		
		aoiLoadLeft.material := aoiLoadRight.material := '';
		aoiLoadLeft.execute := aoiLoadRight.execute := FALSE;
		
		loadStep := 0;
		load := TRUE;
END_CASE

//--------------------------------------------------
IF aoiLoadLeft.recovery THEN //if loading in recovery mode - refill table, resume loading when finished
	aoiLoadLeft.execute := stageEx(
		robot:= robotLeft, 
		aoiTemplate:= aoiTemplateLeft, 
		aoiStaging:= aoiStageLeft, 
		stageStep:= stageStepLeft, 
		includeTop:= TRUE, 
		includeLeft:= TRUE, 
		includeRight:= FALSE, 
		includeBottom:= FALSE, 
		error=> );
ELSE
	//loadLeft.execute := NOT loadLeft.busy AND NOT loadLeft.done;
END_IF
//--------------------------------------------------
IF aoiLoadRight.recovery THEN
	aoiLoadRight.execute := stageEx(
		robot:= robotRight, 
		aoiTemplate:= aoiTemplateRight, 
		aoiStaging:= aoiStageRight, 
		stageStep:= stageStepRight, 
		includeTop:= FALSE, 
		includeLeft:= FALSE, 
		includeRight:= TRUE, 
		includeBottom:= TRUE, 
		error=> );
ELSE
	//loadRight.execute := NOT loadRight.busy AND NOT loadRight.done;
END_IF
//--------------------------------------------------
	
error := aoiLoadLeft.error OR aoiLoadRight.error;
*)
END_METHOD

METHOD PRIVATE loadEx : BOOL
VAR_IN_OUT
	robot : RobotA21;
	aoiLoad : AOI_LoadWoodBunk;
	loadStep : INT;
END_VAR
VAR_INPUT
	pairIndex : INT;
	includeTop, includeLeft, includeRight, includeBottom : BOOL;
END_VAR
VAR_OUTPUT
	error : BOOL;
END_VAR
VAR
	pair : REFERENCE TO PositionMaterials REF= materialsArr[pairIndex];
END_VAR
{warning disable C0371}
IF robot.error THEN
	error := TRUE;
	RETURN;
ELSIF robot.reservation <> sectionID AND_THEN NOT robot.reserve(sectionID) THEN
	RETURN;
ELSIF robot.tool <> sectionID AND_THEN NOT robot.changeEOAT(targetTool := sectionID) THEN
	RETURN;
END_IF

error := aoiLoad.error;

CASE loadStep OF
	0:
		loadStep := Surface.TOP;
	
	Surface.TOP:		
		IF NOT includeTop OR aoiLoad.donePulse THEN
			aoiLoad.execute := FALSE;
			aoiLoad.material := '';
			loadStep := Surface.BOTTOM;
			RETURN;
		END_IF
		
		aoiLoad.surfaceID := Surface.TOP;
		aoiLoad.material := pair.top;
		aoiLoad.suctions := suctionTop;
		aoiLoad.numPads := UPPER_BOUND(suctionTop, 1) - LOWER_BOUND(suctionTop, 1) + 1;
		
		aoiLoad.execute := NOT aoiLoad.busy;
		
	Surface.BOTTOM:
		IF NOT includeBottom OR aoiLoad.donePulse THEN
			aoiLoad.execute := FALSE;
			aoiLoad.material := '';
			loadStep := Surface.LEFT;
			RETURN;
		END_IF
		
		aoiLoad.surfaceID := Surface.BOTTOM;
		aoiLoad.material := pair.bottom;
		aoiLoad.suctions := suctionBottom;
		aoiLoad.numPads := UPPER_BOUND(suctionBottom, 1) - LOWER_BOUND(suctionBottom, 1) + 1;
		
		aoiLoad.execute := NOT aoiLoad.busy;
		
	Surface.LEFT:
		IF NOT includeLeft OR aoiLoad.donePulse THEN
			aoiLoad.execute := FALSE;
			aoiLoad.material := '';
			loadStep := Surface.RIGHT;
			RETURN;
		END_IF
		
		aoiLoad.surfaceID := Surface.LEFT;
		aoiLoad.material := pair.left;
		aoiLoad.suctions := suctionLeft;
		aoiLoad.numPads := UPPER_BOUND(suctionLeft, 1) - LOWER_BOUND(suctionLeft, 1) + 1;
		
		aoiLoad.execute := NOT aoiLoad.busy;
		
	Surface.RIGHT:
		IF NOT includeRight OR aoiLoad.donePulse THEN
			aoiLoad.execute := FALSE;
			aoiLoad.material := '';
			loadStep := COMPLETE;
			RETURN;
		END_IF
		
		aoiLoad.surfaceID := Surface.RIGHT;
		aoiLoad.material := pair.right;
		aoiLoad.suctions := suctionRight;
		aoiLoad.numPads := UPPER_BOUND(suctionRight, 1) - LOWER_BOUND(suctionRight, 1) + 1;
		
		aoiLoad.execute := NOT aoiLoad.busy;
		
	COMPLETE:				
		robot.release(sectionID);
		
		aoiLoad.material := '';
		aoiLoad.execute := FALSE;
		
		loadEx := TRUE;
END_CASE
END_METHOD

METHOD PROTECTED maintenance : BOOL
VAR_INPUT
END_VAR
{warning disable C0371}
//no specific tasks yet, free run and testing
SetSuctions(suctionTop, suctionEnableTop);
SetSuctions(suctionLeft, suctionEnableLeft);
SetSuctions(suctionRight, suctionEnableRight);
SetSuctions(suctionBottom, suctionEnableBottom);

IF robotLeft.Done THEN
	robotLeft.clearCommand();
END_IF

IF robotRight.Done THEN
	robotRight.clearCommand();
END_IF
END_METHOD

METHOD PROTECTED process : BOOL
VAR_INPUT
	auto : BOOL;
END_VAR
VAR_OUTPUT
	error : BOOL;
END_VAR
VAR
	currentPair : REFERENCE TO PositionMaterials REF= materialsArr[iPair];
END_VAR
{warning disable C0371}
CASE step OF
	IDLE:
		IF auto OR_ELSE execute THEN
			step := STAGING;
		END_IF

	LOAD_WB:
		IF
			directionCheckAndSet(conveyorPos, currentPair.position) AND 
			( (auto AND done) OR_ELSE (NOT auto AND execute) )
		THEN
			robotLeft.clearCommand();
			robotRight.clearCommand();
			
			aoiLoadLeft.reset();
			aoiLoadRight.reset();
			
			loadStepLeft := loadStepRight := 0;
			stageStepLeft := stageStepRight := 0;
			
			done := FALSE;
			suctionEnableTop := suctionEnableLeft := suctionEnableRight := suctionEnableBottom := FALSE;
			execute := FALSE;
			
			step := PUSH;
			RETURN;
		END_IF
		
		IF NOT done THEN
			done := load(pairIndex := iPair, error => error);
		END_IF
		
		IF NOT auto THEN
			SetSuctions(suctionTop, suctionEnableTop);
			SetSuctions(suctionLeft, suctionEnableLeft);
			SetSuctions(suctionRight, suctionEnableRight);
			SetSuctions(suctionBottom, suctionEnableBottom);
		END_IF
		
	PUSH:
		IF
			(auto AND latchLeft AND latchRight AND pistonBottom.extended) OR_ELSE
			(NOT auto AND execute)
		THEN
			insertionLeft.stop();
			insertionRight.stop();
			
			latchLeft := latchRight := FALSE;
			execute := FALSE;
			step := STRAP;
			RETURN;
		END_IF
		
		IF NOT validateInsertion(checkTop:= FALSE, checkLeft:= FALSE, checkRight:= FALSE, checkBottom:= FALSE) THEN
			error := TRUE;
			RETURN;
		END_IF
		(*
		IF 
			insertionLeft.sliderPos <> demoHeight/2 //OR 
			//insertionRight.sliderPos <> demoHeight/2 //OR 
			//NOT insertionBottom.contact
		THEN
			insertionLeft.slideAbsolute(demoHeight/2);
			//insertionRight.slideAbsolute(demoHeight/2);
			RETURN;
		END_IF
		*)
		
		IF insertionLeft.Contact THEN
			latchLeft := TRUE;
		ELSIF NOT latchLeft THEN
			insertionLeft.press();
		END_IF
		
		IF insertionRight.Contact THEN
			latchRight := TRUE;
		ELSIF NOT latchRight THEN
			insertionRight.press();
		END_IF
		pistonBottom.extend();
		
	STRAP:	
		strapper.bEnable := TRUE;
		IF strapper.done THEN
			suctionRelease.IN := FALSE;
			step := RELEASE;
			RETURN;
		END_IF
		
		IF suctionRelease.Q THEN
			SetSuctions(suctionTop, FALSE);
			SetSuctions(suctionLeft, FALSE);
			SetSuctions(suctionRight, FALSE);
			SetSuctions(suctionBottom, FALSE);
		ELSIF strapper.atBundleLevel THEN
			suctionRelease.IN := TRUE;
		END_IF
		
		IF strapper.ready THEN
			strapper.strap();
		END_IF
		
		IF execute THEN
			suctionRelease.IN := FALSE;
			execute := FALSE;
			step := RELEASE;
		END_IF
		
	RELEASE: //release command		
		//insertionLeft.slideAbsolute(0);
		//insertionRight.slideAbsolute(0);
		
		insertionLeft.release();
		insertionRight.release();
		pistonBottom.retract();
		
		IF 
			(insertionLeft.screw.AtHome AND insertionRight.screw.AtHome AND pistonBottom.retracted) OR
			execute
		THEN
			execute := FALSE;
			step := COMPLETE;
		END_IF
	
	COMPLETE:
		//reset everything
		iPair := (iPair + 1) MOD GVL.maxPairs;
		step := IDLE;
		
		process := TRUE;
END_CASE
END_METHOD

METHOD PROTECTED ps_AbortCondition : BOOL
VAR_INPUT
END_VAR
{warning disable C0371}
ps_AbortCondition :=
	insertionLeft.error OR 
	insertionRight.error OR 
	robotLeft.error OR 
	robotRight.error OR
	strapper.error;
END_METHOD

METHOD PROTECTED ps_Aborted : BOOL
VAR_INPUT
END_VAR
ps_Aborted := TRUE;
END_METHOD

METHOD PROTECTED ps_Aborting : BOOL
VAR_INPUT
END_VAR
{warning disable C0371}
insertionLeft.stop();
insertionRight.stop();
pistonBottom.stop();

aoiLoadLeft.reset();
aoiLoadRight.reset();

aoiStageLeft.reset();
aoiStageRight.reset();

robotLeft.clearCommand();
robotRight.clearCommand();

//stop conveyors

ps_Aborting :=
	NOT insertionLeft.active AND
	NOT insertionRight.active AND
	NOT pistonBottom.busy AND
	NOT robotLeft.Busy AND
	NOT robotRight.Busy;
END_METHOD

METHOD PROTECTED ps_Clearing : BOOL
VAR_INPUT
END_VAR
{warning disable C0371}
insertionLeft.reset();
insertionRight.reset();

ps_Clearing := 
	NOT insertionLeft.error AND
	NOT insertionRight.error AND
	NOT strapper.error AND
	NOT robotLeft.error AND
	NOT robotRight.error;
END_METHOD

METHOD PROTECTED ps_Complete : BOOL
VAR_INPUT
END_VAR
ps_Complete := TRUE;
END_METHOD

METHOD PROTECTED ps_Completing : BOOL
VAR_INPUT
END_VAR
ps_Completing := NOT occupied;
END_METHOD

METHOD PROTECTED ps_Execute : BOOL
VAR_INPUT
END_VAR
VAR_OUTPUT
	error : BOOL;
END_VAR
END_METHOD

METHOD PROTECTED ps_Held : BOOL
VAR_INPUT
END_VAR
ps_Held := NOT hold;
END_METHOD

METHOD PROTECTED ps_HoldCondition : BOOL
VAR_INPUT
END_VAR
END_METHOD

METHOD PROTECTED ps_Holding : BOOL
VAR_INPUT
END_VAR
{warning disable C0371}
insertionLeft.stop();
insertionRight.stop();
pistonBottom.stop();
//set robot to pause

ps_Holding :=
	NOT insertionLeft.active AND
	NOT insertionRight.active;
END_METHOD

METHOD PROTECTED ps_Idle : BOOL
VAR_INPUT
END_VAR
ps_Idle := execute;
execute := FALSE;
END_METHOD

METHOD PROTECTED ps_Resetting : BOOL
VAR_INPUT
END_VAR
{warning disable C0371}
insertionLeft.reset();
insertionRight.reset();

ps_Resetting := 
	reset AND
	NOT insertionLeft.error AND
	NOT insertionRight.error AND
	NOT strapper.error AND
	NOT robotLeft.error AND
	NOT robotRight.error;
END_METHOD

METHOD PROTECTED ps_Starting : BOOL
VAR_INPUT
END_VAR
{warning disable C0371}
robotLeft.clearCommand();
robotRight.clearCommand();

insertionLeft.homingSequence();
insertionRight.homingSequence();
pistonBottom.retract();

ps_Starting := 
	insertionLeft.screw.HomeSet AND 
	insertionRight.screw.HomeSet AND 
	pistonBottom.retracted;
END_METHOD

METHOD PROTECTED ps_StopCondition : BOOL
VAR_INPUT
END_VAR
ps_StopCondition := 
	stop;
END_METHOD

METHOD PROTECTED ps_Stopped : BOOL
VAR_INPUT
END_VAR
ps_Stopped := TRUE;
END_METHOD

METHOD PROTECTED ps_Stopping : BOOL
VAR_INPUT
END_VAR
{warning disable C0371}
insertionLeft.stop();
insertionRight.stop();
pistonBottom.stop();

aoiLoadLeft.reset();
aoiLoadRight.reset();

aoiStageLeft.reset();
aoiStageRight.reset();

robotLeft.clearCommand();
robotRight.clearCommand();

//stop conveyors

ps_Stopping :=
	NOT insertionLeft.active AND
	NOT insertionRight.active AND
	NOT pistonBottom.busy AND
	NOT robotLeft.Busy AND
	NOT robotRight.Busy;
END_METHOD

METHOD PROTECTED ps_SuspendCondition : BOOL
VAR_INPUT
END_VAR
END_METHOD

METHOD PROTECTED ps_Suspended : BOOL
VAR_INPUT
END_VAR
ps_Suspended := NOT ps_SuspendCondition();
END_METHOD

METHOD PROTECTED ps_Suspending : BOOL
VAR_INPUT
END_VAR
ps_Suspending := TRUE;
END_METHOD

METHOD PROTECTED ps_Unholding : BOOL
VAR_INPUT
END_VAR
ps_Unholding := TRUE;
END_METHOD

METHOD PROTECTED ps_Unsuspending : BOOL
VAR_INPUT
END_VAR
ps_Unsuspending := TRUE;
END_METHOD

METHOD PROTECTED stage : BOOL
VAR_OUTPUT
	error : BOOL;
END_VAR
{warning disable C0371}

(*
this method only exists to call stageEx() for both robots
*)
(*
stage := leftDone AND rightDone;

IF NOT leftDone THEN
	leftDone := stageEx(
		robot:= robotLeft, 
		aoiTemplate:= aoiTemplateLeft, 
		aoiStaging:= aoiStageLeft, 
		stageStep:= stageStepLeft, 
		//iSlot:= iSlotLeft, 
		includeTop:= TRUE, 
		includeLeft:= TRUE, 
		includeRight:= FALSE, 
		includeBottom:= FALSE, 
		error=> );
END_IF

IF NOT rightDone THEN
	rightDone := stageEx(
		robot:= robotRight, 
		aoiTemplate:= aoiTemplateRight, 
		aoiStaging:= aoiStageRight, 
		stageStep:= stageStepRight, 
		//iSlot:= iSlotRight, 
		includeTop:= FALSE, 
		includeLeft:= FALSE, 
		includeRight:= TRUE, 
		includeBottom:= TRUE, 
		error=> );
END_IF
*)

stage := 
	stageEx(
		robot:= robotLeft, 
		aoiTemplate:= aoiTemplateLeft, 
		aoiStaging:= aoiStageLeft, 
		stageStep:= stageStepLeft, 
		includeTop:= TRUE, 
		includeLeft:= TRUE, 
		includeRight:= FALSE, 
		includeBottom:= FALSE, 
		error=> )
	AND
	stageEx(
		robot:= robotRight, 
		aoiTemplate:= aoiTemplateRight, 
		aoiStaging:= aoiStageRight, 
		stageStep:= stageStepRight, 
		includeTop:= FALSE, 
		includeLeft:= FALSE, 
		includeRight:= TRUE, 
		includeBottom:= TRUE, 
		error=> );
END_METHOD

